C07227=1039.766,-84.411,-76.368,168.767,36.325,156.840
C07228=1039.759,-84.660,-76.358,168.765,36.326,156.840
C07229=1039.754,-84.910,-76.347,168.762,36.326,156.840
C07230=1039.747,-85.160,-76.336,168.760,36.326,156.840
C07231=1039.741,-85.409,-76.325,168.757,36.326,156.840
C07232=1039.734,-85.659,-76.314,168.755,36.326,156.840
C07233=1039.728,-85.909,-76.304,168.752,36.326,156.840
C07234=1039.722,-86.158,-76.293,168.750,36.327,156.840
C07235=1039.716,-86.408,-76.282,168.747,36.327,156.840
C07236=1039.709,-86.658,-76.271,168.745,36.327,156.840
C07237=1039.704,-86.908,-76.261,168.742,36.327,156.840
C07238=1039.698,-87.158,-76.250,168.740,36.327,156.840
C07239=1039.691,-87.407,-76.240,168.737,36.327,156.840
C07240=1039.685,-87.656,-76.229,168.735,36.327,156.840
C07241=1039.679,-87.907,-76.218,168.732,36.327,156.840
C07242=1039.673,-88.156,-76.207,168.730,36.327,156.840
C07243=1039.667,-88.405,-76.196,168.727,36.328,156.840
C07244=1039.660,-88.655,-76.186,168.725,36.328,156.840
C07245=1039.654,-88.905,-76.176,168.722,36.328,156.840
C07246=1039.649,-89.155,-76.165,168.720,36.328,156.840
C07247=1039.642,-89.405,-76.154,168.717,36.328,156.840
C07248=1039.636,-89.654,-76.143,168.715,36.328,156.840
C07249=1039.630,-89.904,-76.132,168.712,36.328,156.840
C07250=1039.624,-90.153,-76.123,168.710,36.328,156.840
C07251=1039.618,-90.404,-76.111,168.707,36.328,156.840
C07252=1039.611,-90.653,-76.101,168.705,36.329,156.841
C07253=1039.605,-90.902,-76.090,168.702,36.329,156.841
C07254=1039.600,-91.152,-76.080,168.700,36.329,156.841
C07255=1039.593,-91.402,-76.069,168.697,36.329,156.841
C07256=1039.587,-91.652,-76.059,168.695,36.330,156.841
C07257=1039.581,-91.901,-76.048,168.692,36.330,156.841
C07258=1039.575,-92.151,-76.038,168.690,36.330,156.841
C07259=1039.569,-92.401,-76.027,168.687,36.330,156.841
C07260=1039.562,-92.650,-76.017,168.685,36.330,156.841
C07261=1039.557,-92.901,-76.006,168.682,36.330,156.841
C07262=1039.550,-93.150,-75.996,168.680,36.330,156.841
C07263=1039.545,-93.399,-75.985,168.678,36.331,156.841
C07264=1039.539,-93.650,-75.975,168.676,36.331,156.841
C07265=1039.532,-93.899,-75.965,168.673,36.331,156.841
C07266=1039.526,-94.149,-75.954,168.671,36.331,156.841
C07267=1039.520,-94.399,-75.944,168.668,36.331,156.841
C07268=1039.515,-94.648,-75.933,168.666,36.331,156.841
C07269=1039.508,-94.897,-75.923,168.663,36.331,156.841
C07270=1039.502,-95.148,-75.912,168.661,36.332,156.841
C07271=1039.496,-95.398,-75.901,168.658,36.332,156.841
C07272=1039.490,-95.647,-75.891,168.656,36.332,156.841
C07273=1039.484,-95.897,-75.881,168.653,36.333,156.841
C07274=1039.478,-96.146,-75.871,168.651,36.333,156.841
C07275=1039.472,-96.396,-75.861,168.648,36.333,156.841
C07276=1039.466,-96.645,-75.850,168.646,36.333,156.841
C07277=1039.460,-96.896,-75.840,168.643,36.333,156.841
C07278=1039.454,-97.146,-75.829,168.641,36.333,156.841
C07279=1039.448,-97.395,-75.819,168.638,36.333,156.841
C07280=1039.442,-97.645,-75.809,168.636,36.334,156.842
C07281=1039.436,-97.895,-75.799,168.633,36.334,156.842
C07282=1039.430,-98.144,-75.789,168.630,36.335,156.842
C07283=1039.423,-98.394,-75.779,168.628,36.335,156.842
C07284=1039.417,-98.644,-75.768,168.625,36.335,156.842
C07285=1039.411,-98.894,-75.758,168.623,36.335,156.842
C07286=1039.404,-99.143,-75.748,168.620,36.336,156.842
C07287=1039.399,-99.393,-75.738,168.618,36.336,156.842
C07288=1039.392,-99.680,-75.727,168.615,36.336,156.842
C07289=1039.384,-99.967,-75.715,168.612,36.337,156.842
C07290=1039.378,-100.255,-75.703,168.609,36.337,156.842
C07291=1039.371,-100.541,-75.692,168.606,36.338,156.842
C07292=1039.364,-100.791,-75.681,168.603,36.338,156.842
C07293=1039.358,-101.041,-75.671,168.601,36.338,156.842
C07294=1039.352,-101.291,-75.662,168.598,36.338,156.842
C07295=1039.346,-101.540,-75.651,168.596,36.339,156.842
C07296=1039.340,-101.790,-75.641,168.593,36.340,156.843
C07297=1039.334,-102.040,-75.632,168.591,36.340,156.843
C07298=1039.328,-102.289,-75.621,168.589,36.340,156.843
C07299=1039.322,-102.539,-75.611,168.586,36.340,156.843
C07300=1039.316,-102.789,-75.602,168.584,36.341,156.843
C07301=1039.310,-103.038,-75.591,168.581,36.341,156.843
C07302=1039.303,-103.288,-75.582,168.579,36.342,156.843
C07303=1039.298,-103.538,-75.572,168.576,36.341,156.843
C07304=1039.291,-103.787,-75.561,168.574,36.342,156.843
C07305=1039.285,-104.037,-75.552,168.571,36.343,156.843
C07306=1039.279,-104.287,-75.542,168.568,36.343,156.843
C07307=1039.274,-104.537,-75.532,168.566,36.343,156.843
C07308=1039.267,-104.786,-75.522,168.563,36.343,156.843
C07309=1039.261,-105.036,-75.512,168.561,36.344,156.843
C07310=1039.255,-105.286,-75.503,168.558,36.345,156.844
C07311=1039.249,-105.536,-75.492,168.556,36.345,156.844
C07312=1039.243,-105.786,-75.483,168.553,36.345,156.844
C07313=1039.237,-106.035,-75.472,168.550,36.345,156.844
C07314=1039.231,-106.285,-75.463,168.548,36.346,156.844
C07315=1039.224,-106.535,-75.453,168.545,36.347,156.844
C07316=1039.219,-106.785,-75.443,168.543,36.347,156.844
C07317=1039.213,-107.034,-75.434,168.540,36.347,156.844
C07318=1039.207,-107.284,-75.424,168.538,36.348,156.844
C07319=1039.200,-107.533,-75.414,168.535,36.348,156.844
C07320=1039.194,-107.783,-75.404,168.532,36.349,156.844
C07321=1039.188,-108.033,-75.395,168.530,36.349,156.844
C07322=1039.182,-108.283,-75.384,168.528,36.350,156.844
C07323=1039.176,-108.533,-75.375,168.526,36.350,156.844
C07324=1039.170,-108.783,-75.365,168.523,36.350,156.845
C07325=1039.164,-109.033,-75.356,168.520,36.351,156.845
C07326=1039.158,-109.282,-75.346,168.518,36.352,156.845
C07327=1039.152,-109.532,-75.337,168.515,36.352,156.845
C07328=1039.146,-109.781,-75.327,168.513,36.352,156.845
C07329=1039.140,-110.031,-75.318,168.510,36.353,156.845
C07330=1039.134,-110.281,-75.308,168.507,36.354,156.845
C07331=1039.127,-110.531,-75.299,168.505,36.354,156.845
C07332=1039.121,-110.780,-75.289,168.502,36.354,156.845
///RCONF 1,0,0,0,1,0,0,0,0,0,0,0,0,0,0,0,0,0,0,0,0,0,0,0
C07333=1039.115,-111.030,-75.280,168.499,36.355,156.845
C07334=1039.109,-111.280,-75.270,168.497,36.356,156.845
C07335=1039.103,-111.530,-75.260,168.494,36.356,156.846
C07336=1039.097,-111.780,-75.251,168.492,36.356,156.846
C07337=1039.090,-112.029,-75.241,168.489,36.357,156.846
C07338=1039.086,-112.279,-75.232,168.486,36.357,156.846
C07339=1039.079,-112.529,-75.222,168.484,36.358,156.846
C07340=1039.073,-112.778,-75.212,168.481,36.359,156.846
C07341=1039.067,-113.028,-75.203,168.479,36.359,156.846
C07342=1039.061,-113.278,-75.193,168.477,36.359,156.846
C07343=1039.055,-113.528,-75.184,168.474,36.360,156.846
C07344=1039.049,-113.778,-75.174,168.472,36.361,156.846
C07345=1039.043,-114.027,-75.165,168.469,36.361,156.847
C07346=1039.037,-114.276,-75.155,168.467,36.362,156.847
C07347=1039.031,-114.526,-75.146,168.464,36.362,156.847
C07348=1039.025,-114.777,-75.137,168.461,36.363,156.847
C07349=1039.019,-115.027,-75.127,168.459,36.363,156.847
C07350=1039.012,-115.276,-75.118,168.456,36.364,156.847
C07351=1039.007,-115.525,-75.109,168.453,36.365,156.847
C07352=1038.999,-115.812,-75.098,168.450,36.365,156.847
C07353=1038.993,-116.098,-75.087,168.447,36.366,156.847
C07354=1038.985,-116.385,-75.077,168.444,36.367,156.847
C07355=1038.979,-116.671,-75.066,168.441,36.367,156.848
C07356=1038.972,-116.921,-75.057,168.439,36.368,156.848
C07357=1038.967,-117.170,-75.048,168.436,36.368,156.848
C07358=1038.961,-117.420,-75.038,168.434,36.369,156.848
C07359=1038.954,-117.670,-75.028,168.432,36.370,156.848
C07360=1038.949,-117.920,-75.020,168.429,36.370,156.848
C07361=1038.942,-118.169,-75.011,168.427,36.371,156.848
C07362=1038.936,-118.419,-75.001,168.424,36.372,156.848
C07363=1038.930,-118.669,-74.993,168.421,36.372,156.848
C07364=1038.924,-118.919,-74.983,168.419,36.373,156.849
C07365=1038.918,-119.168,-74.974,168.416,36.374,156.849
C07366=1038.912,-119.418,-74.964,168.413,36.374,156.849
C07367=1038.906,-119.668,-74.955,168.411,36.375,156.849
C07368=1038.900,-119.918,-74.946,168.408,36.376,156.849
C07369=1038.894,-120.167,-74.937,168.405,36.376,156.849
C07370=1038.888,-120.417,-74.928,168.403,36.377,156.849
C07371=1038.882,-120.667,-74.919,168.400,36.378,156.849
C07372=1038.876,-120.917,-74.909,168.398,36.378,156.849
C07373=1038.870,-121.167,-74.901,168.395,36.379,156.850
C07374=1038.864,-121.416,-74.892,168.393,36.379,156.850
C07375=1038.858,-121.666,-74.883,168.391,36.380,156.850
C07376=1038.852,-121.916,-74.874,168.388,36.381,156.850
C07377=1038.846,-122.165,-74.864,168.385,36.381,156.850
C07378=1038.840,-122.416,-74.855,168.383,36.382,156.850
C07379=1038.834,-122.665,-74.847,168.380,36.383,156.850
C07380=1038.828,-122.915,-74.838,168.377,36.384,156.851
C07381=1038.822,-123.165,-74.828,168.375,36.385,156.851
C07382=1038.816,-123.414,-74.819,168.372,36.385,156.851
C07383=1038.810,-123.664,-74.811,168.369,36.386,156.851
C07384=1038.803,-123.914,-74.801,168.367,36.387,156.851
C07385=1038.798,-124.163,-74.793,168.364,36.387,156.851
C07386=1038.792,-124.413,-74.783,168.361,36.388,156.851
C07387=1038.785,-124.663,-74.775,168.359,36.389,156.851
C07388=1038.780,-124.912,-74.766,168.357,36.389,156.851
C07389=1038.774,-125.163,-74.757,168.354,36.391,156.852
C07390=1038.767,-125.412,-74.748,168.352,36.391,156.852
C07391=1038.762,-125.662,-74.739,168.349,36.392,156.852
C07392=1038.756,-125.912,-74.730,168.346,36.392,156.852
C07393=1038.750,-126.161,-74.722,168.344,36.393,156.852
C07394=1038.744,-126.412,-74.713,168.341,36.394,156.852
C07395=1038.738,-126.661,-74.704,168.338,36.395,156.852
C07396=1038.732,-126.911,-74.696,168.336,36.396,156.853
C07397=1038.725,-127.161,-74.686,168.333,36.396,156.853
C07398=1038.720,-127.410,-74.678,168.330,36.397,156.853
C07399=1038.714,-127.661,-74.669,168.328,36.398,156.853
C07400=1038.708,-127.910,-74.660,168.326,36.399,156.853
C07401=1038.703,-128.160,-74.650,168.324,36.399,156.853
C07402=1038.698,-128.409,-74.640,168.321,36.399,156.853
C07403=1038.695,-128.658,-74.630,168.318,36.398,156.853
C07404=1038.692,-128.909,-74.618,168.316,36.397,156.853
C07405=1038.690,-129.158,-74.607,168.314,36.396,156.853
C07406=1038.689,-129.409,-74.594,168.312,36.394,156.852
C07407=1038.689,-129.658,-74.581,168.311,36.391,156.852
C07408=1038.690,-129.909,-74.567,168.308,36.388,156.851
C07409=1038.690,-130.159,-74.553,168.307,36.384,156.851
C07410=1038.692,-130.409,-74.538,168.306,36.381,156.850
C07411=1038.695,-130.659,-74.523,168.304,36.377,156.849
C07412=1038.698,-130.909,-74.507,168.303,36.372,156.849
C07413=1038.703,-131.160,-74.490,168.301,36.367,156.848
C07414=1038.707,-131.409,-74.473,168.301,36.361,156.847
C07415=1038.713,-131.660,-74.455,168.300,36.355,156.846
C07416=1038.372,-131.683,-74.721,168.252,36.557,156.880
C07417=1038.366,-131.435,-74.739,168.253,36.564,156.881
C07418=1038.360,-131.184,-74.756,168.254,36.569,156.882
C07419=1038.356,-130.934,-74.773,168.255,36.574,156.883
C07420=1038.353,-130.683,-74.788,168.256,36.579,156.883
C07421=1038.350,-130.434,-74.805,168.258,36.584,156.884
C07422=1038.348,-130.184,-74.819,168.259,36.587,156.885
C07423=1038.347,-129.933,-74.834,168.261,36.591,156.885
C07424=1038.346,-129.683,-74.847,168.263,36.593,156.886
C07425=1038.347,-129.433,-74.860,168.264,36.596,156.886
C07426=1038.349,-129.184,-74.873,168.266,36.598,156.887
C07427=1038.350,-128.934,-74.885,168.269,36.600,156.887
C07428=1038.352,-128.683,-74.896,168.271,36.601,156.887
C07429=1038.357,-128.434,-74.907,168.273,36.601,156.887
C07430=1038.361,-128.184,-74.917,168.276,36.602,156.887
C07431=1038.365,-127.934,-74.926,168.278,36.601,156.887
C07432=1038.371,-127.685,-74.935,168.281,36.601,156.887
C07433=1038.377,-127.435,-74.944,168.283,36.600,156.887
C07434=1038.383,-127.185,-74.953,168.286,36.599,156.887
C07435=1038.389,-126.935,-74.962,168.288,36.598,156.887
C07436=1038.395,-126.686,-74.970,168.291,36.597,156.887
C07437=1038.401,-126.436,-74.979,168.293,36.597,156.886
C07438=1038.407,-126.185,-74.988,168.296,36.596,156.886
C07439=1038.413,-125.937,-74.997,168.299,36.595,156.886
C07440=1038.419,-125.686,-75.005,168.301,36.594,156.886
C07441=1038.425,-125.437,-75.015,168.304,36.593,156.886
C07442=1038.431,-125.187,-75.023,168.307,36.593,156.886
C07443=1038.437,-124.937,-75.032,168.309,36.592,156.886
C07444=1038.443,-124.688,-75.041,168.312,36.591,156.885
C07445=1038.450,-124.438,-75.050,168.315,36.590,156.885
C07446=1038.455,-124.188,-75.059,168.317,36.589,156.885
C07447=1038.461,-123.939,-75.068,168.320,36.589,156.885
C07448=1038.467,-123.688,-75.077,168.322,36.588,156.885
C07449=1038.474,-123.439,-75.086,168.324,36.587,156.885
C07450=1038.479,-123.189,-75.094,168.327,36.587,156.885
C07451=1038.485,-122.939,-75.104,168.330,36.585,156.885
C07452=1038.491,-122.689,-75.113,168.332,36.585,156.884
C07453=1038.497,-122.440,-75.122,168.335,36.584,156.884
C07454=1038.504,-122.190,-75.131,168.338,36.583,156.884
C07455=1038.509,-121.940,-75.140,168.340,36.583,156.884
C07456=1038.515,-121.691,-75.149,168.343,36.582,156.884
C07457=1038.521,-121.440,-75.158,168.346,36.581,156.884
C07458=1038.527,-121.190,-75.167,168.348,36.581,156.884
C07459=1038.533,-120.942,-75.176,168.351,36.580,156.884
C07460=1038.539,-120.691,-75.185,168.354,36.579,156.884
C07461=1038.545,-120.441,-75.194,168.355,36.578,156.883
C07462=1038.551,-120.192,-75.204,168.358,36.577,156.883
C07463=1038.557,-119.942,-75.212,168.361,36.577,156.883
C07464=1038.563,-119.692,-75.222,168.363,36.576,156.883
C07465=1038.570,-119.443,-75.231,168.366,36.575,156.883
C07466=1038.575,-119.193,-75.239,168.369,36.575,156.883
C07467=1038.581,-118.943,-75.249,168.371,36.574,156.883
C07468=1038.587,-118.693,-75.259,168.374,36.573,156.883
C07469=1038.593,-118.443,-75.267,168.377,36.573,156.882
C07470=1038.599,-118.194,-75.277,168.379,36.572,156.882
C07471=1038.605,-117.944,-75.286,168.382,36.571,156.882
C07472=1038.612,-117.694,-75.295,168.385,36.571,156.882
C07473=1038.618,-117.444,-75.304,168.387,36.570,156.882
C07474=1038.623,-117.195,-75.313,168.390,36.569,156.882
C07475=1038.630,-116.945,-75.323,168.392,36.569,156.882
C07476=1038.636,-116.695,-75.332,168.394,36.568,156.882
C07477=1038.642,-116.409,-75.343,168.397,36.567,156.882
C07478=1038.650,-116.122,-75.354,168.400,36.567,156.881
C07479=1038.657,-115.836,-75.364,168.403,36.566,156.881
C07480=1038.663,-115.550,-75.375,168.406,36.565,156.881
C07481=1038.670,-115.300,-75.384,168.409,36.565,156.881
C07482=1038.676,-115.051,-75.393,168.412,36.564,156.881
C07483=1038.682,-114.801,-75.403,168.414,36.563,156.881
C07484=1038.688,-114.550,-75.412,168.417,36.563,156.881
C07485=1038.694,-114.301,-75.421,168.420,36.562,156.881
C07486=1038.700,-114.052,-75.431,168.422,36.562,156.881
C07487=1038.706,-113.802,-75.440,168.425,36.561,156.880
C07488=1038.712,-113.552,-75.450,168.427,36.560,156.880
C07489=1038.718,-113.302,-75.459,168.430,36.560,156.880
C07490=1038.724,-113.052,-75.469,168.433,36.560,156.880
C07491=1038.730,-112.803,-75.478,168.434,36.559,156.880
C07492=1038.736,-112.553,-75.488,168.437,36.558,156.880
C07493=1038.742,-112.304,-75.497,168.440,36.558,156.880
C07494=1038.748,-112.054,-75.507,168.442,36.557,156.880
C07495=1038.753,-111.803,-75.516,168.445,36.556,156.880
C07496=1038.760,-111.553,-75.526,168.447,36.556,156.880
C07497=1038.766,-111.304,-75.535,168.450,36.556,156.880
C07498=1038.772,-111.054,-75.545,168.453,36.555,156.880
C07499=1038.778,-110.804,-75.554,168.455,36.554,156.879
C07500=1038.784,-110.555,-75.564,168.458,36.554,156.879
C07501=1038.790,-110.305,-75.573,168.461,36.553,156.879
C07502=1038.796,-110.055,-75.583,168.463,36.553,156.879
C07503=1038.802,-109.805,-75.592,168.466,36.552,156.879
C07504=1038.809,-109.556,-75.603,168.468,36.552,156.879
C07505=1038.815,-109.306,-75.612,168.471,36.551,156.879
C07506=1038.821,-109.057,-75.622,168.474,36.550,156.879
///RCONF 1,0,0,0,0,0,0,0,0,0,0,0,0,0,0,0,0,0,0,0,0,0,0,0
C07507=1038.827,-108.807,-75.631,168.476,36.550,156.879
C07508=1038.833,-108.557,-75.641,168.479,36.550,156.879
C07509=1038.840,-108.307,-75.651,168.481,36.549,156.879
C07510=1038.845,-108.057,-75.661,168.483,36.548,156.878
C07511=1038.851,-107.807,-75.670,168.486,36.548,156.878
C07512=1038.857,-107.558,-75.680,168.488,36.548,156.878
C07513=1038.864,-107.308,-75.689,168.491,36.547,156.878
C07514=1038.870,-107.058,-75.699,168.494,36.546,156.878
C07515=1038.876,-106.810,-75.709,168.496,36.546,156.878
C07516=1038.882,-106.560,-75.718,168.499,36.546,156.878
C07517=1038.887,-106.310,-75.729,168.501,36.545,156.878
C07518=1038.893,-106.060,-75.738,168.504,36.544,156.878
C07519=1038.900,-105.810,-75.748,168.507,36.544,156.878
C07520=1038.906,-105.560,-75.757,168.509,36.544,156.878
C07521=1038.911,-105.311,-75.768,168.512,36.543,156.878
C07522=1038.918,-105.061,-75.778,168.514,36.543,156.878
C07523=1038.924,-104.811,-75.787,168.517,36.542,156.877
C07524=1038.930,-104.561,-75.797,168.520,36.542,156.877
C07525=1038.936,-104.312,-75.808,168.522,36.542,156.877
C07526=1038.942,-104.062,-75.817,168.525,36.541,156.877
C07527=1038.948,-103.812,-75.827,168.527,36.541,156.877
C07528=1038.954,-103.562,-75.836,168.530,36.540,156.877
C07529=1038.960,-103.313,-75.847,168.532,36.540,156.877
C07530=1038.966,-103.063,-75.857,168.535,36.540,156.877
C07531=1038.972,-102.813,-75.866,168.537,36.539,156.877
C07532=1038.979,-102.564,-75.877,168.539,36.539,156.877
C07533=1038.985,-102.313,-75.887,168.542,36.538,156.877
C07534=1038.991,-102.064,-75.897,168.544,36.538,156.877
C07535=1038.997,-101.814,-75.906,168.547,36.538,156.877
C07536=1039.003,-101.564,-75.917,168.550,36.537,156.877
C07537=1039.009,-101.314,-75.927,168.552,36.537,156.877
C07538=1039.016,-101.065,-75.937,168.555,36.536,156.876
C07539=1039.022,-100.816,-75.947,168.557,36.536,156.876
C07540=1039.027,-100.565,-75.957,168.560,36.536,156.876
C07541=1039.035,-100.279,-75.969,168.563,36.535,156.876
C07542=1039.042,-99.991,-75.980,168.566,36.534,156.876
C07543=1039.049,-99.704,-75.992,168.569,36.534,156.876
C07544=1039.055,-99.417,-76.003,168.572,36.534,156.876
C07545=1039.062,-99.167,-76.013,168.574,36.534,156.876
C07546=1039.068,-98.917,-76.024,168.577,36.533,156.876
C07547=1039.074,-98.668,-76.034,168.579,36.532,156.876
C07548=1039.081,-98.418,-76.043,168.582,36.532,156.876
C07549=1039.086,-98.168,-76.054,168.585,36.532,156.876
C07550=1039.092,-97.919,-76.064,168.587,36.532,156.876
C07551=1039.099,-97.669,-76.073,168.590,36.531,156.875
C07552=1039.105,-97.419,-76.085,168.592,36.531,156.875
C07553=1039.111,-97.169,-76.094,168.595,36.531,156.875
C07554=1039.117,-96.920,-76.105,168.597,36.531,156.875
C07555=1039.123,-96.670,-76.115,168.600,36.531,156.875
C07556=1039.129,-96.420,-76.126,168.602,36.530,156.875
C07557=1039.135,-96.171,-76.136,168.605,36.530,156.875
C07558=1039.141,-95.921,-76.146,168.607,36.530,156.875
C07559=1039.146,-95.672,-76.157,168.609,36.529,156.875
C07560=1039.153,-95.421,-76.167,168.611,36.529,156.875
C07561=1039.159,-95.172,-76.178,168.614,36.529,156.875
C07562=1039.165,-94.922,-76.188,168.617,36.529,156.875
C07563=1039.171,-94.672,-76.198,168.619,36.529,156.875
C07564=1039.177,-94.423,-76.209,168.622,36.529,156.875
C07565=1039.183,-94.174,-76.219,168.624,36.528,156.875
C07566=1039.189,-93.923,-76.230,168.627,36.528,156.875
C07567=1039.196,-93.674,-76.240,168.629,36.528,156.875
C07568=1039.201,-93.423,-76.250,168.632,36.527,156.875
C07569=1039.207,-93.174,-76.261,168.634,36.527,156.875
C07570=1039.213,-92.925,-76.271,168.637,36.527,156.875
C07571=1039.219,-92.675,-76.282,168.639,36.527,156.875
C07572=1039.226,-92.425,-76.292,168.642,36.527,156.875
C07573=1039.231,-92.175,-76.303,168.644,36.527,156.875
C07574=1039.238,-91.926,-76.313,168.647,36.526,156.875
C07575=1039.243,-91.676,-76.324,168.649,36.526,156.875
C07576=1039.250,-91.426,-76.335,168.652,36.526,156.875
C07577=1039.256,-91.177,-76.345,168.654,36.525,156.874
C07578=1039.262,-90.927,-76.356,168.657,36.525,156.874
C07579=1039.268,-90.677,-76.366,168.659,36.525,156.874
C07580=1039.274,-90.427,-76.377,168.662,36.525,156.874
C07581=1039.280,-90.178,-76.388,168.664,36.525,156.874
C07582=1039.287,-89.929,-76.398,168.667,36.525,156.874
C07583=1039.292,-89.678,-76.408,168.669,36.525,156.874
C07584=1039.299,-89.429,-76.419,168.672,36.524,156.874
C07585=1039.305,-89.179,-76.430,168.674,36.524,156.874
C07586=1039.311,-88.930,-76.440,168.677,36.524,156.874
C07587=1039.318,-88.680,-76.451,168.680,36.523,156.874
C07588=1039.323,-88.430,-76.461,168.682,36.523,156.874
C07589=1039.329,-88.180,-76.472,168.685,36.523,156.874
C07590=1039.335,-87.931,-76.482,168.687,36.523,156.874
C07591=1039.342,-87.681,-76.494,168.690,36.523,156.874
C07592=1039.348,-87.432,-76.504,168.692,36.523,156.874
C07593=1039.354,-87.182,-76.515,168.695,36.523,156.874
C07594=1039.360,-86.932,-76.526,168.697,36.523,156.874
C07595=1039.366,-86.682,-76.536,168.700,36.522,156.874
C07596=1039.372,-86.433,-76.547,168.702,36.522,156.874
C07597=1039.379,-86.182,-76.558,168.705,36.522,156.874
C07598=1039.385,-85.933,-76.568,168.707,36.522,156.874
C07599=1039.391,-85.683,-76.579,168.710,36.521,156.874
C07600=1039.397,-85.434,-76.590,168.712,36.521,156.874
C07601=1039.404,-85.184,-76.600,168.715,36.521,156.874
C07602=1039.410,-84.934,-76.612,168.717,36.521,156.874
C07603=1039.416,-84.685,-76.623,168.720,36.521,156.874
C07604=1039.422,-84.436,-76.633,168.722,36.521,156.874
C07605=1039.429,-84.150,-76.645,168.725,36.521,156.874
C07606=1039.437,-83.865,-76.657,168.728,36.521,156.874
C07607=1039.444,-83.580,-76.669,168.731,36.520,156.874
C07608=1039.450,-83.295,-76.683,168.733,36.520,156.874
C07609=1039.457,-83.046,-76.693,168.736,36.520,156.874
C07610=1039.463,-82.796,-76.705,168.738,36.520,156.874
C07611=1039.469,-82.546,-76.715,168.741,36.520,156.874
C07612=1039.476,-82.296,-76.726,168.742,36.519,156.873
C07613=1039.482,-82.047,-76.737,168.745,36.519,156.873
C07614=1039.488,-81.797,-76.748,168.747,36.519,156.873
C07615=1039.495,-81.548,-76.758,168.750,36.519,156.873
C07616=1039.501,-81.297,-76.770,168.752,36.519,156.873
C07617=1039.507,-81.048,-76.781,168.755,36.519,156.873
C07618=1039.513,-80.799,-76.791,168.757,36.519,156.873
C07619=1039.519,-80.548,-76.802,168.760,36.519,156.873
C07620=1039.525,-80.299,-76.813,168.762,36.519,156.873
C07621=1039.532,-80.049,-76.824,168.765,36.519,156.873
C07622=1039.538,-79.800,-76.835,168.767,36.518,156.873
C07623=1039.545,-79.550,-76.847,168.770,36.518,156.873
C07624=1039.550,-79.301,-76.857,168.772,36.518,156.873
C07625=1039.557,-79.050,-76.869,168.775,36.518,156.873
C07626=1039.563,-78.801,-76.880,168.777,36.518,156.873
C07627=1039.569,-78.551,-76.891,168.780,36.518,156.873
C07628=1039.575,-78.302,-76.902,168.782,36.518,156.873
C07629=1039.581,-78.052,-76.914,168.784,36.518,156.873
C07630=1039.587,-77.802,-76.924,168.787,36.518,156.873
C07631=1039.593,-77.552,-76.936,168.789,36.518,156.873
C07632=1039.600,-77.303,-76.947,168.792,36.518,156.873
C07633=1039.606,-77.053,-76.958,168.794,36.518,156.873
C07634=1039.612,-76.804,-76.969,168.797,36.518,156.873
C07635=1039.619,-76.553,-76.980,168.799,36.518,156.873
C07636=1039.625,-76.305,-76.992,168.802,36.518,156.873
C07637=1039.631,-76.054,-77.003,168.804,36.518,156.873
C07638=1039.637,-75.805,-77.014,168.806,36.518,156.873
C07639=1039.643,-75.555,-77.026,168.809,36.518,156.873
C07640=1039.649,-75.306,-77.037,168.811,36.518,156.873
C07641=1039.655,-75.056,-77.048,168.814,36.519,156.873
C07642=1039.662,-74.806,-77.060,168.816,36.519,156.873
C07643=1039.668,-74.557,-77.071,168.819,36.519,156.873
C07644=1039.674,-74.306,-77.082,168.821,36.519,156.873
C07645=1039.680,-74.058,-77.094,168.823,36.519,156.873
C07646=1039.686,-73.807,-77.105,168.826,36.519,156.873
C07647=1039.692,-73.558,-77.116,168.828,36.519,156.873
C07648=1039.699,-73.308,-77.128,168.831,36.519,156.873
C07649=1039.704,-73.058,-77.139,168.833,36.519,156.873
C07650=1039.711,-72.809,-77.151,168.835,36.519,156.873
C07651=1039.717,-72.559,-77.162,168.838,36.519,156.873
C07652=1039.723,-72.310,-77.174,168.840,36.519,156.873
C07653=1039.729,-72.059,-77.186,168.843,36.519,156.873
C07654=1039.735,-71.811,-77.197,168.846,36.520,156.874
C07655=1039.741,-71.560,-77.209,168.848,36.520,156.874
C07656=1039.747,-71.311,-77.220,168.851,36.520,156.874
C07657=1039.753,-71.061,-77.231,168.853,36.520,156.874
C07658=1039.759,-70.811,-77.244,168.856,36.520,156.874
C07659=1039.765,-70.562,-77.255,168.858,36.521,156.874
C07660=1039.772,-70.312,-77.267,168.860,36.521,156.874
C07661=1039.777,-70.063,-77.278,168.863,36.521,156.874
C07662=1039.783,-69.813,-77.290,168.865,36.521,156.874
C07663=1039.790,-69.563,-77.301,168.867,36.521,156.874
C07664=1039.796,-69.314,-77.313,168.870,36.521,156.874
C07665=1039.802,-69.064,-77.324,168.872,36.521,156.874
C07666=1039.807,-68.814,-77.336,168.875,36.521,156.874
C07667=1039.814,-68.565,-77.348,168.877,36.522,156.874
C07668=1039.820,-68.315,-77.360,168.879,36.522,156.874
C07669=1039.827,-68.032,-77.373,168.882,36.522,156.874
C07670=1039.834,-67.750,-77.386,168.885,36.523,156.874
C07671=1039.841,-67.467,-77.400,168.887,36.523,156.874
C07672=1039.848,-67.184,-77.413,168.890,36.523,156.874
C07673=1039.855,-66.934,-77.425,168.892,36.523,156.874
C07674=1039.860,-66.685,-77.436,168.895,36.523,156.874
C07675=1039.866,-66.435,-77.448,168.897,36.523,156.874
C07676=1039.873,-66.185,-77.460,168.900,36.523,156.874
C07677=1039.878,-65.936,-77.472,168.902,36.523,156.874
C07678=1039.885,-65.686,-77.484,168.904,36.524,156.874
C07679=1039.891,-65.436,-77.495,168.907,36.524,156.874
C07680=1039.897,-65.187,-77.506,168.909,36.524,156.874
C07681=1039.903,-64.937,-77.519,168.911,36.524,156.874
C07682=1039.910,-64.688,-77.531,168.914,36.524,156.874
C07683=1039.916,-64.437,-77.542,168.916,36.524,156.874
C07684=1039.921,-64.188,-77.554,168.918,36.524,156.874
C07685=1039.928,-63.939,-77.566,168.921,36.525,156.875
C07686=1039.935,-63.689,-77.578,168.923,36.525,156.875
C07687=1039.941,-63.439,-77.589,168.925,36.525,156.875
C07688=1039.946,-63.190,-77.602,168.928,36.526,156.875
C07689=1039.953,-62.940,-77.614,168.930,36.526,156.875
C07690=1039.960,-62.691,-77.626,168.933,36.526,156.875
C07691=1039.965,-62.441,-77.638,168.935,36.526,156.875
C07692=1039.971,-62.191,-77.649,168.937,36.526,156.875
C07693=1039.978,-61.942,-77.661,168.940,36.526,156.875
C07694=1039.984,-61.692,-77.673,168.942,36.526,156.875
C07695=1039.990,-61.442,-77.685,168.944,36.527,156.875
C07696=1039.997,-61.193,-77.697,168.947,36.527,156.875
C07697=1040.003,-60.944,-77.709,168.949,36.527,156.875
C07698=1040.009,-60.693,-77.721,168.951,36.528,156.875
C07699=1040.015,-60.444,-77.733,168.954,36.528,156.875
C07700=1040.022,-60.194,-77.745,168.956,36.528,156.875
C07701=1040.028,-59.944,-77.757,168.958,36.528,156.875
C07702=1040.035,-59.695,-77.769,168.961,36.528,156.875
C07703=1040.041,-59.446,-77.781,168.963,36.528,156.875
C07704=1040.046,-59.196,-77.793,168.966,36.529,156.875
C07705=1040.053,-58.946,-77.805,168.969,36.529,156.875
C07706=1040.059,-58.696,-77.817,168.971,36.529,156.875
C07707=1040.065,-58.446,-77.829,168.973,36.530,156.875
C07708=1040.072,-58.197,-77.841,168.976,36.530,156.875
C07709=1040.079,-57.947,-77.853,168.978,36.530,156.875
C07710=1040.084,-57.698,-77.865,168.980,36.530,156.875
C07711=1040.091,-57.448,-77.877,168.983,36.530,156.875
C07712=1040.097,-57.199,-77.889,168.985,36.530,156.875
C07713=1040.103,-56.949,-77.902,168.987,36.531,156.876
C07714=1040.110,-56.699,-77.914,168.990,36.531,156.876
C07715=1040.116,-56.450,-77.926,168.992,36.531,156.876
C07716=1040.122,-56.200,-77.938,168.994,36.532,156.876
C07717=1040.129,-55.935,-77.951,168.997,36.532,156.876
C07718=1040.136,-55.671,-77.963,168.999,36.532,156.876
C07719=1040.143,-55.405,-77.977,169.002,36.532,156.876
C07720=1040.150,-55.141,-77.990,169.004,36.532,156.876
C07721=1040.156,-54.891,-78.002,169.007,36.533,156.876
C07722=1040.162,-54.641,-78.015,169.009,36.533,156.876
C07723=1040.169,-54.392,-78.027,169.011,36.533,156.876
C07724=1040.175,-54.142,-78.039,169.014,36.533,156.876
C07725=1040.181,-53.892,-78.051,169.016,36.533,156.876
C07726=1040.188,-53.643,-78.063,169.018,36.533,156.876
C07727=1040.194,-53.393,-78.076,169.021,36.534,156.876
C07728=1040.201,-53.143,-78.088,169.023,36.534,156.876
C07729=1040.207,-52.894,-78.099,169.025,36.535,156.876
C07730=1040.213,-52.644,-78.112,169.028,36.535,156.876
C07731=1040.220,-52.394,-78.124,169.030,36.535,156.876
C07732=1040.226,-52.145,-78.137,169.032,36.535,156.876
C07733=1040.233,-51.879,-78.149,169.035,36.535,156.876
C07734=1040.239,-51.613,-78.162,169.037,36.536,156.876
C07735=1040.247,-51.346,-78.176,169.040,36.536,156.876
C07736=1040.253,-51.080,-78.189,169.042,36.536,156.876
C07737=1040.260,-50.831,-78.201,169.044,36.537,156.877
C07738=1040.266,-50.581,-78.214,169.047,36.537,156.877
C07739=1040.272,-50.332,-78.226,169.049,36.537,156.877
C07740=1040.278,-50.082,-78.239,169.051,36.537,156.877
C07741=1040.284,-49.832,-78.251,169.053,36.538,156.877
C07742=1040.291,-49.583,-78.264,169.057,36.539,156.877
C07743=1040.297,-49.333,-78.276,169.059,36.539,156.877
C07744=1040.303,-49.083,-78.289,169.061,36.539,156.877
C07745=1040.309,-48.834,-78.302,169.063,36.539,156.877
C07746=1040.316,-48.584,-78.314,169.066,36.540,156.877
C07747=1040.322,-48.335,-78.327,169.068,36.541,156.877
C07748=1040.328,-48.085,-78.340,169.070,36.541,156.877
C07749=1040.334,-47.835,-78.353,169.072,36.541,156.877
C07750=1040.341,-47.586,-78.364,169.075,36.542,156.878
C07751=1040.347,-47.337,-78.378,169.077,36.542,156.878
C07752=1040.353,-47.087,-78.390,169.079,36.542,156.878
C07753=1040.359,-46.837,-78.403,169.081,36.542,156.878
C07754=1040.366,-46.588,-78.416,169.084,36.543,156.878
C07755=1040.372,-46.337,-78.428,169.086,36.544,156.878
C07756=1040.378,-46.087,-78.441,169.088,36.544,156.878
C07757=1040.384,-45.838,-78.454,169.090,36.544,156.878
C07758=1040.391,-45.589,-78.466,169.093,36.545,156.878
C07759=1040.397,-45.339,-78.480,169.095,36.545,156.878
C07760=1040.403,-45.089,-78.492,169.097,36.546,156.878
C07761=1040.409,-44.840,-78.505,169.099,36.546,156.878
C07762=1040.416,-44.591,-78.517,169.102,36.546,156.878
C07763=1040.422,-44.341,-78.530,169.104,36.547,156.878
C07764=1040.428,-44.091,-78.543,169.106,36.547,156.878
C07765=1040.434,-43.842,-78.556,169.109,36.548,156.879
C07766=1040.441,-43.593,-78.568,169.112,36.548,156.879
C07767=1040.447,-43.342,-78.581,169.114,36.548,156.879
C07768=1040.454,-43.093,-78.595,169.116,36.549,156.879
C07769=1040.459,-42.843,-78.607,169.118,36.550,156.879
C07770=1040.466,-42.594,-78.620,169.120,36.550,156.879
C07771=1040.472,-42.344,-78.632,169.123,36.550,156.879
C07772=1040.479,-42.095,-78.646,169.125,36.551,156.879
C07773=1040.484,-41.845,-78.658,169.127,36.551,156.879
C07774=1040.491,-41.596,-78.671,169.129,36.551,156.879
C07775=1040.497,-41.346,-78.685,169.132,36.552,156.879
C07776=1040.504,-41.096,-78.697,169.134,36.552,156.879
C07777=1040.510,-40.847,-78.710,169.136,36.553,156.879
C07778=1040.516,-40.597,-78.723,169.138,36.553,156.880
C07779=1040.522,-40.348,-78.736,169.140,36.553,156.880
C07780=1040.529,-40.097,-78.749,169.143,36.554,156.880
C07781=1040.536,-39.848,-78.762,169.145,36.555,156.880
C07782=1040.542,-39.599,-78.775,169.147,36.555,156.880
C07783=1040.548,-39.349,-78.788,169.149,36.555,156.880
C07784=1040.554,-39.100,-78.801,169.152,36.556,156.880
C07785=1040.561,-38.850,-78.814,169.154,36.556,156.880
C07786=1040.567,-38.600,-78.827,169.157,36.557,156.880
C07787=1040.573,-38.351,-78.840,169.159,36.557,156.880
C07788=1040.579,-38.101,-78.854,169.161,36.558,156.880
C07789=1040.585,-37.851,-78.866,169.163,36.558,156.881
C07790=1040.592,-37.602,-78.879,169.166,36.558,156.881
C07791=1040.598,-37.352,-78.893,169.168,36.559,156.881
C07792=1040.604,-37.102,-78.906,169.170,36.560,156.881
C07793=1040.610,-36.853,-78.919,169.172,36.560,156.881
C07794=1040.617,-36.604,-78.932,169.174,36.561,156.881
C07795=1040.623,-36.355,-78.945,169.177,36.562,156.881
C07796=1040.629,-36.104,-78.958,169.179,36.562,156.881
C07797=1040.636,-35.824,-78.973,169.181,36.562,156.881
C07798=1040.643,-35.542,-78.988,169.184,36.563,156.881
C07799=1040.651,-35.261,-79.003,169.186,36.564,156.881
C07800=1040.657,-34.980,-79.018,169.188,36.564,156.882
C07801=1040.664,-34.730,-79.032,169.191,36.565,156.882
C07802=1040.670,-34.481,-79.045,169.193,36.566,156.882
C07803=1040.676,-34.232,-79.058,169.196,36.566,156.882
C07804=1040.683,-33.982,-79.072,169.198,36.567,156.882
C07805=1040.689,-33.732,-79.084,169.200,36.567,156.882
C07806=1040.695,-33.483,-79.098,169.202,36.567,156.882
C07807=1040.701,-33.233,-79.111,169.205,36.568,156.882
C07808=1040.708,-32.983,-79.124,169.207,36.569,156.882
C07809=1040.714,-32.734,-79.138,169.209,36.569,156.883
C07810=1040.720,-32.485,-79.151,169.211,36.570,156.883
C07811=1040.727,-32.235,-79.165,169.213,36.571,156.883
C07812=1040.733,-31.986,-79.178,169.215,36.571,156.883
C07813=1040.740,-31.736,-79.191,169.218,36.571,156.883
C07814=1040.745,-31.486,-79.204,169.220,36.572,156.883
C07815=1040.752,-31.236,-79.218,169.222,36.573,156.883
C07816=1040.758,-30.987,-79.231,169.224,36.573,156.883
C07817=1040.764,-30.738,-79.244,169.226,36.574,156.883
C07818=1040.771,-30.488,-79.258,169.228,36.574,156.883
C07819=1040.777,-30.239,-79.271,169.230,36.574,156.883
C07820=1040.783,-29.989,-79.285,169.234,36.575,156.884
C07821=1040.790,-29.739,-79.298,169.236,36.576,156.884
C07822=1040.796,-29.490,-79.312,169.238,36.576,156.884
C07823=1040.803,-29.240,-79.325,169.240,36.577,156.884
C07824=1040.809,-28.991,-79.338,169.242,36.578,156.884
C07825=1040.815,-28.741,-79.352,169.244,36.578,156.884
C07826=1040.822,-28.491,-79.366,169.246,36.578,156.884
C07827=1040.828,-28.242,-79.379,169.249,36.579,156.884
C07828=1040.834,-27.993,-79.392,169.251,36.580,156.884
C07829=1040.841,-27.743,-79.406,169.253,36.580,156.884
C07830=1040.847,-27.494,-79.419,169.255,36.581,156.885
C07831=1040.854,-27.244,-79.433,169.257,36.581,156.885
C07832=1040.860,-26.994,-79.446,169.259,36.582,156.885
C07833=1040.866,-26.745,-79.460,169.261,36.583,156.885
C07834=1040.873,-26.495,-79.474,169.263,36.583,156.885
C07835=1040.879,-26.246,-79.488,169.267,36.584,156.885
C07836=1040.884,-25.997,-79.502,169.269,36.585,156.885
C07837=1040.891,-25.747,-79.515,169.271,36.585,156.885
C07838=1040.897,-25.497,-79.529,169.273,36.586,156.886
C07839=1040.904,-25.247,-79.543,169.275,36.587,156.886
C07840=1040.910,-24.998,-79.556,169.277,36.587,156.886
C07841=1040.916,-24.749,-79.571,169.279,36.588,156.886
C07842=1040.922,-24.499,-79.584,169.281,36.589,156.886
C07843=1040.929,-24.250,-79.598,169.283,36.589,156.886
C07844=1040.935,-23.999,-79.612,169.285,36.590,156.886
C07845=1040.941,-23.750,-79.625,169.288,36.590,156.886
C07846=1040.947,-23.501,-79.639,169.290,36.591,156.886
C07847=1040.953,-23.251,-79.653,169.292,36.592,156.887
C07848=1040.960,-23.002,-79.667,169.294,36.592,156.887
C07849=1040.966,-22.752,-79.680,169.297,36.593,156.887
C07850=1040.972,-22.503,-79.695,169.299,36.594,156.887
C07851=1040.979,-22.253,-79.708,169.301,36.594,156.887
C07852=1040.985,-22.003,-79.722,169.303,36.595,156.887
C07853=1040.991,-21.753,-79.736,169.305,36.596,156.887
C07854=1040.998,-21.505,-79.750,169.307,36.596,156.887
C07855=1041.004,-21.255,-79.764,169.309,36.597,156.888
C07856=1041.010,-21.005,-79.777,169.311,36.597,156.888
C07857=1041.017,-20.756,-79.792,169.314,36.598,156.888
C07858=1041.023,-20.506,-79.806,169.316,36.599,156.888
C07859=1041.030,-20.256,-79.819,169.318,36.599,156.888
C07860=1041.035,-20.007,-79.833,169.320,36.600,156.888
C07861=1041.043,-19.725,-79.849,169.322,36.601,156.888
C07862=1041.050,-19.444,-79.865,169.324,36.601,156.888
C07863=1041.057,-19.161,-79.880,169.328,36.603,156.889
C07864=1041.064,-18.880,-79.896,169.330,36.603,156.889
C07865=1041.070,-18.630,-79.910,169.332,36.604,156.889
C07866=1041.077,-18.381,-79.925,169.334,36.604,156.889
C07867=1041.083,-18.131,-79.938,169.336,36.605,156.889
C07868=1041.089,-17.881,-79.952,169.338,36.606,156.889
C07869=1041.096,-17.632,-79.966,169.340,36.606,156.889
C07870=1041.102,-17.383,-79.980,169.343,36.607,156.889
C07871=1041.109,-17.133,-79.995,169.345,36.608,156.890
C07872=1041.115,-16.884,-80.008,169.347,36.608,156.890
C07873=1041.121,-16.634,-80.023,169.349,36.609,156.890
C07874=1041.128,-16.385,-80.036,169.351,36.610,156.890
C07875=1041.134,-16.135,-80.050,169.353,36.610,156.890
C07876=1041.140,-15.886,-80.064,169.356,36.611,156.890
C07877=1041.147,-15.636,-80.078,169.358,36.611,156.890
C07878=1041.153,-15.386,-80.093,169.360,36.612,156.890
C07879=1041.160,-15.137,-80.106,169.362,36.613,156.890
C07880=1041.166,-14.887,-80.121,169.364,36.614,156.891
C07881=1041.172,-14.638,-80.135,169.366,36.615,156.891
C07882=1041.179,-14.388,-80.149,169.368,36.615,156.891
C07883=1041.184,-14.139,-80.163,169.370,36.616,156.891
C07884=1041.191,-13.889,-80.178,169.372,36.617,156.891
C07885=1041.198,-13.640,-80.193,169.374,36.617,156.891
C07886=1041.203,-13.390,-80.206,169.376,36.618,156.891
C07887=1041.210,-13.140,-80.221,169.378,36.619,156.892
C07888=1041.216,-12.891,-80.235,169.381,36.620,156.892
C07889=1041.222,-12.642,-80.250,169.383,36.620,156.892
C07890=1041.228,-12.392,-80.265,169.385,36.621,156.892
C07891=1041.235,-12.143,-80.278,169.387,36.622,156.892
C07892=1041.241,-11.893,-80.293,169.389,36.623,156.892
C07893=1041.247,-11.643,-80.307,169.391,36.623,156.892
C07894=1041.254,-11.394,-80.321,169.393,36.624,156.893
C07895=1041.260,-11.144,-80.336,169.395,36.625,156.893
C07896=1041.266,-10.895,-80.350,169.397,36.625,156.893
C07897=1041.273,-10.645,-80.364,169.399,36.627,156.893
C07898=1041.279,-10.396,-80.379,169.401,36.627,156.893
C07899=1041.285,-10.146,-80.393,169.403,36.628,156.893
C07900=1041.292,-9.897,-80.407,169.406,36.629,156.893
C07901=1041.298,-9.647,-80.422,169.408,36.629,156.893
C07902=1041.304,-9.398,-80.437,169.410,36.630,156.894
C07903=1041.311,-9.148,-80.450,169.412,36.631,156.894
C07904=1041.317,-8.899,-80.465,169.414,36.632,156.894
C07905=1041.323,-8.650,-80.480,169.416,36.632,156.894
C07906=1041.330,-8.400,-80.494,169.418,36.633,156.894
C07907=1041.336,-8.150,-80.509,169.420,36.634,156.894
C07908=1041.342,-7.901,-80.523,169.422,36.635,156.895
C07909=1041.348,-7.651,-80.538,169.424,36.636,156.895
C07910=1041.355,-7.402,-80.552,169.426,36.636,156.895
C07911=1041.361,-7.153,-80.566,169.428,36.637,156.895
C07912=1041.367,-6.903,-80.581,169.431,36.637,156.895
C07913=1041.374,-6.654,-80.596,169.433,36.639,156.895
C07914=1041.381,-6.404,-80.611,169.435,36.639,156.895
C07915=1041.386,-6.154,-80.624,169.437,36.640,156.895
C07916=1041.393,-5.905,-80.639,169.439,36.641,156.896
C07917=1041.400,-5.655,-80.654,169.441,36.641,156.896
C07918=1041.405,-5.406,-80.668,169.443,36.642,156.896
C07919=1041.412,-5.157,-80.683,169.445,36.643,156.896
C07920=1041.419,-4.907,-80.698,169.447,36.644,156.896
C07921=1041.425,-4.657,-80.712,169.449,36.644,156.896
C07922=1041.431,-4.407,-80.727,169.451,36.645,156.896
C07923=1041.437,-4.158,-80.741,169.453,36.646,156.897
C07924=1041.444,-3.909,-80.756,169.456,36.647,156.897
C07925=1041.451,-3.626,-80.772,169.459,36.648,156.897
C07926=1041.459,-3.343,-80.789,169.461,36.648,156.897
C07927=1041.466,-3.058,-80.806,169.463,36.649,156.897
C07928=1041.473,-2.775,-80.823,169.465,36.651,156.897
C07929=1041.479,-2.526,-80.837,169.467,36.651,156.898
C07930=1041.485,-2.276,-80.852,169.469,36.652,156.898
C07931=1041.491,-2.027,-80.867,169.471,36.653,156.898
C07932=1041.498,-1.777,-80.882,169.473,36.654,156.898
C07933=1041.503,-1.528,-80.897,169.476,36.655,156.898
C07934=1041.510,-1.278,-80.912,169.478,36.656,156.898
C07935=1041.516,-1.029,-80.927,169.480,36.656,156.899
C07936=1041.523,-0.779,-80.942,169.482,36.658,156.899
C07937=1041.529,-0.531,-80.957,169.484,36.658,156.899
C07938=1041.535,-0.281,-80.972,169.486,36.659,156.899
C07939=1041.541,-0.031,-80.987,169.488,36.660,156.899
C07940=1041.547,0.219,-81.002,169.489,36.661,156.899
C07941=1041.553,0.468,-81.017,169.491,36.662,156.899
C07942=1041.559,0.717,-81.032,169.493,36.663,156.900
C07943=1041.566,0.967,-81.047,169.496,36.663,156.900
C07944=1041.572,1.217,-81.062,169.498,36.664,156.900
C07945=1041.578,1.466,-81.077,169.500,36.665,156.900
C07946=1041.585,1.716,-81.092,169.502,36.666,156.900
C07947=1041.591,1.965,-81.106,169.504,36.667,156.901
C07948=1041.597,2.214,-81.121,169.506,36.668,156.901
C07949=1041.604,2.464,-81.137,169.508,36.668,156.901
C07950=1041.610,2.713,-81.152,169.510,36.670,156.901
C07951=1041.616,2.963,-81.167,169.512,36.670,156.901
C07952=1041.622,3.212,-81.181,169.514,36.671,156.901
C07953=1041.629,3.461,-81.196,169.517,36.672,156.902
C07954=1041.635,3.711,-81.211,169.518,36.673,156.902
C07955=1041.642,3.960,-81.227,169.520,36.674,156.902
C07956=1041.647,4.210,-81.242,169.522,36.675,156.902
C07957=1041.654,4.460,-81.257,169.524,36.675,156.902
C07958=1041.660,4.709,-81.272,169.526,36.677,156.902
C07959=1041.666,4.959,-81.287,169.528,36.677,156.902
C07960=1041.673,5.207,-81.303,169.530,36.678,156.903
C07961=1041.679,5.457,-81.317,169.532,36.679,156.903
C07962=1041.685,5.707,-81.332,169.534,36.680,156.903
C07963=1041.692,5.956,-81.347,169.537,36.680,156.903
C07964=1041.698,6.205,-81.363,169.539,36.682,156.903
C07965=1041.705,6.455,-81.378,169.541,36.682,156.903
C07966=1041.711,6.705,-81.393,169.542,36.683,156.904
C07967=1041.718,6.954,-81.408,169.544,36.684,156.904
C07968=1041.723,7.204,-81.424,169.546,36.685,156.904
C07969=1041.730,7.453,-81.439,169.548,36.686,156.904
C07970=1041.736,7.703,-81.454,169.550,36.687,156.904
C07971=1041.742,7.951,-81.469,169.552,36.687,156.904
C07972=1041.749,8.201,-81.484,169.554,36.689,156.905
C07973=1041.755,8.451,-81.499,169.557,36.689,156.905
C07974=1041.761,8.700,-81.514,169.559,36.690,156.905
C07975=1041.768,8.949,-81.530,169.561,36.691,156.905
C07976=1041.775,9.199,-81.545,169.563,36.692,156.905
C07977=1041.780,9.449,-81.560,169.564,36.692,156.905
C07978=1041.787,9.698,-81.576,169.566,36.694,156.906
C07979=1041.793,9.948,-81.591,169.568,36.694,156.906
C07980=1041.800,10.197,-81.607,169.570,36.695,156.906
C07981=1041.806,10.446,-81.622,169.572,36.696,156.906
C07982=1041.813,10.696,-81.636,169.574,36.697,156.906
C07983=1041.819,10.945,-81.652,169.576,36.698,156.906
C07984=1041.826,11.195,-81.667,169.579,36.699,156.906
C07985=1041.833,11.444,-81.683,169.581,36.699,156.907
C07986=1041.838,11.694,-81.698,169.583,36.700,156.907
C07987=1041.845,11.943,-81.713,169.585,36.701,156.907
C07988=1041.851,12.192,-81.729,169.586,36.702,156.907
C07989=1041.859,12.478,-81.747,169.589,36.703,156.907
C07990=1041.866,12.764,-81.764,169.591,36.704,156.907
C07991=1041.874,13.049,-81.781,169.593,36.705,156.908
C07992=1041.881,13.334,-81.799,169.595,36.706,156.908
C07993=1041.887,13.584,-81.814,169.598,36.707,156.908
C07994=1041.893,13.833,-81.830,169.600,36.708,156.908
C07995=1041.900,14.083,-81.845,169.602,36.708,156.908
C07996=1041.906,14.332,-81.861,169.604,36.709,156.908
C07997=1041.913,14.581,-81.876,169.606,36.710,156.909
C07998=1041.919,14.831,-81.892,169.607,36.711,156.909
C07999=1041.925,15.080,-81.908,169.609,36.712,156.909
C08000=1041.931,15.330,-81.923,169.611,36.713,156.909
C08001=1041.938,15.579,-81.939,169.613,36.714,156.909
C08002=1041.944,15.828,-81.954,169.616,36.715,156.910
C08003=1041.950,16.078,-81.970,169.618,36.716,156.910
C08004=1041.957,16.327,-81.986,169.620,36.717,156.910
C08005=1041.962,16.577,-82.001,169.621,36.718,156.910
C08006=1041.969,16.826,-82.017,169.623,36.719,156.910
C08007=1041.976,17.076,-82.032,169.625,36.720,156.910
C08008=1041.982,17.325,-82.048,169.627,36.721,156.911
C08009=1041.989,17.575,-82.064,169.629,36.721,156.911
C08010=1041.994,17.824,-82.080,169.631,36.723,156.911
C08011=1042.001,18.074,-82.095,169.634,36.723,156.911
C08012=1042.008,18.323,-82.111,169.635,36.725,156.911
C08013=1042.013,18.573,-82.126,169.637,36.725,156.911
C08014=1042.020,18.822,-82.142,169.639,36.726,156.912
C08015=1042.026,19.071,-82.158,169.641,36.727,156.912
C08016=1042.032,19.321,-82.173,169.643,36.728,156.912
C08017=1042.039,19.570,-82.189,169.645,36.729,156.912
C08018=1042.045,19.819,-82.205,169.647,36.730,156.912
C08019=1042.052,20.069,-82.221,169.648,36.731,156.913
C08020=1042.058,20.319,-82.237,169.651,36.732,156.913
C08021=1042.065,20.568,-82.252,169.653,36.733,156.913
C08022=1042.071,20.817,-82.269,169.655,36.734,156.913
C08023=1042.077,21.066,-82.284,169.657,36.735,156.913
C08024=1042.083,21.316,-82.300,169.659,36.736,156.913
C08025=1042.090,21.565,-82.316,169.660,36.737,156.914
C08026=1042.096,21.814,-82.332,169.662,36.738,156.914
C08027=1042.102,22.064,-82.348,169.664,36.738,156.914
C08028=1042.109,22.314,-82.364,169.666,36.740,156.914
C08029=1042.115,22.563,-82.380,169.669,36.740,156.914
C08030=1042.121,22.813,-82.395,169.671,36.742,156.915
C08031=1042.127,23.062,-82.412,169.672,36.742,156.915
C08032=1042.134,23.311,-82.427,169.674,36.743,156.915
C08033=1042.140,23.560,-82.444,169.676,36.744,156.915
C08034=1042.147,23.809,-82.459,169.678,36.745,156.915
C08035=1042.153,24.060,-82.475,169.680,36.746,156.915
C08036=1042.159,24.309,-82.491,169.681,36.747,156.916
C08037=1042.165,24.558,-82.507,169.684,36.748,156.916
C08038=1042.171,24.808,-82.523,169.686,36.749,156.916
C08039=1042.178,25.057,-82.539,169.688,36.750,156.916
C08040=1042.185,25.307,-82.556,169.690,36.751,156.916
C08041=1042.191,25.556,-82.571,169.692,36.752,156.917
C08042=1042.197,25.805,-82.587,169.693,36.753,156.917
C08043=1042.204,26.054,-82.603,169.695,36.754,156.917
C08044=1042.210,26.304,-82.619,169.697,36.755,156.917
C08045=1042.216,26.554,-82.636,169.699,36.756,156.917
C08046=1042.223,26.803,-82.651,169.702,36.757,156.917
C08047=1042.229,27.053,-82.667,169.704,36.758,156.918
C08048=1042.235,27.302,-82.683,169.705,36.759,156.918
C08049=1042.241,27.551,-82.699,169.707,36.760,156.918
C08050=1042.248,27.801,-82.716,169.709,36.760,156.918
C08051=1042.255,28.050,-82.731,169.711,36.762,156.918
C08052=1042.261,28.299,-82.748,169.713,36.763,156.919
C08053=1042.268,28.586,-82.766,169.715,36.764,156.919
C08054=1042.275,28.872,-82.786,169.718,36.765,156.919
C08055=1042.282,29.160,-82.804,169.720,36.766,156.919
C08056=1042.290,29.446,-82.822,169.722,36.767,156.919
C08057=1042.296,29.695,-82.839,169.724,36.769,156.920
C08058=1042.302,29.945,-82.855,169.725,36.769,156.920
C08059=1042.308,30.194,-82.871,169.727,36.770,156.920
C08060=1042.315,30.444,-82.887,169.729,36.772,156.920
C08061=1042.321,30.693,-82.904,169.731,36.772,156.920
C08062=1042.327,30.942,-82.921,169.734,36.774,156.921
C08063=1042.333,31.191,-82.937,169.735,36.774,156.921
C08064=1042.340,31.441,-82.953,169.737,36.775,156.921
C08065=1042.346,31.690,-82.969,169.739,36.777,156.921
C08066=1042.352,31.940,-82.985,169.741,36.777,156.921
C08067=1042.358,32.189,-83.002,169.743,36.779,156.922
C08068=1042.365,32.438,-83.019,169.744,36.780,156.922
C08069=1042.372,32.688,-83.035,169.746,36.780,156.922
C08070=1042.378,32.937,-83.051,169.749,36.782,156.922
C08071=1042.384,33.187,-83.067,169.751,36.782,156.922
C08072=1042.390,33.436,-83.084,169.753,36.784,156.923
C08073=1042.396,33.686,-83.100,169.754,36.785,156.923
C08074=1042.402,33.934,-83.117,169.756,36.785,156.923
C08075=1042.410,34.184,-83.133,169.758,36.787,156.923
C08076=1042.416,34.433,-83.149,169.760,36.787,156.923
C08077=1042.422,34.683,-83.165,169.762,36.789,156.924
C08078=1042.428,34.933,-83.182,169.764,36.790,156.924
C08079=1042.434,35.182,-83.199,169.766,36.790,156.924
C08080=1042.441,35.431,-83.215,169.768,36.792,156.924
C08081=1042.448,35.681,-83.231,169.770,36.792,156.924
C08082=1042.454,35.930,-83.248,169.771,36.794,156.924
C08083=1042.460,36.179,-83.265,169.773,36.795,156.925
C08084=1042.466,36.429,-83.281,169.775,36.795,156.925
C08085=1042.472,36.678,-83.297,169.777,36.797,156.925
C08086=1042.479,36.927,-83.314,169.779,36.797,156.925
C08087=1042.486,37.177,-83.330,169.781,36.799,156.925
C08088=1042.492,37.426,-83.347,169.783,36.800,156.926
C08089=1042.498,37.675,-83.363,169.785,36.800,156.926
C08090=1042.505,37.925,-83.380,169.787,36.802,156.926
C08091=1042.511,38.174,-83.397,169.788,36.803,156.926
C08092=1042.517,38.423,-83.414,169.790,36.804,156.926
C08093=1042.523,38.673,-83.430,169.792,36.805,156.927
C08094=1042.529,38.922,-83.446,169.795,36.806,156.927
C08095=1042.536,39.172,-83.464,169.797,36.807,156.927
C08096=1042.542,39.421,-83.480,169.798,36.808,156.927
C08097=1042.548,39.670,-83.496,169.800,36.809,156.927
C08098=1042.554,39.920,-83.514,169.802,36.810,156.928
C08099=1042.560,40.169,-83.530,169.804,36.811,156.928
C08100=1042.566,40.418,-83.547,169.805,36.812,156.928
C08101=1042.573,40.668,-83.564,169.807,36.814,156.928
C08102=1042.579,40.917,-83.581,169.810,36.814,156.928
C08103=1042.586,41.167,-83.598,169.812,36.815,156.929
C08104=1042.592,41.416,-83.615,169.813,36.817,156.929
C08105=1042.598,41.665,-83.631,169.815,36.818,156.929
C08106=1042.605,41.915,-83.647,169.817,36.819,156.929
C08107=1042.611,42.164,-83.664,169.819,36.820,156.930
C08108=1042.617,42.414,-83.681,169.820,36.821,156.930
C08109=1042.624,42.663,-83.698,169.822,36.822,156.930
C08110=1042.630,42.912,-83.714,169.825,36.823,156.930
C08111=1042.636,43.161,-83.732,169.827,36.824,156.930
C08112=1042.643,43.410,-83.749,169.828,36.825,156.930
C08113=1042.649,43.660,-83.766,169.830,36.826,156.931
C08114=1042.655,43.909,-83.783,169.832,36.827,156.931
C08115=1042.661,44.159,-83.799,169.834,36.829,156.931
C08116=1042.667,44.408,-83.817,169.835,36.830,156.931
C08117=1042.674,44.695,-83.836,169.838,36.831,156.932
C08118=1042.681,44.980,-83.856,169.840,36.832,156.932
C08119=1042.688,45.268,-83.875,169.842,36.834,156.932
C08120=1042.695,45.554,-83.894,169.844,36.835,156.932
C08121=1042.701,45.804,-83.912,169.846,36.836,156.933
C08122=1042.708,46.053,-83.929,169.848,36.837,156.933
C08123=1042.713,46.302,-83.946,169.850,36.838,156.933
C08124=1042.720,46.552,-83.963,169.852,36.839,156.933
C08125=1042.726,46.801,-83.981,169.854,36.840,156.933
C08126=1042.732,47.051,-83.997,169.856,36.842,156.934
C08127=1042.739,47.299,-84.014,169.857,36.843,156.934
C08128=1042.745,47.549,-84.032,169.859,36.844,156.934
C08129=1042.751,47.798,-84.048,169.861,36.845,156.934
C08130=1042.758,48.048,-84.066,169.864,36.846,156.935
C08131=1042.763,48.297,-84.083,169.865,36.847,156.935
C08132=1042.770,48.546,-84.101,169.867,36.849,156.935
C08133=1042.776,48.796,-84.117,169.869,36.850,156.935
C08134=1042.781,49.045,-84.134,169.870,36.850,156.935
C08135=1042.788,49.294,-84.152,169.872,36.852,156.936
C08136=1042.794,49.544,-84.168,169.874,36.853,156.936
C08137=1042.800,49.793,-84.186,169.877,36.854,156.936
C08138=1042.807,50.042,-84.203,169.878,36.855,156.936
C08139=1042.813,50.291,-84.220,169.880,36.856,156.937
C08140=1042.819,50.540,-84.238,169.882,36.857,156.937
C08141=1042.826,50.791,-84.254,169.884,36.859,156.937
C08142=1042.831,51.040,-84.272,169.885,36.860,156.937
C08143=1042.838,51.289,-84.289,169.887,36.860,156.937
C08144=1042.844,51.538,-84.306,169.889,36.862,156.938
C08145=1042.850,51.787,-84.324,169.891,36.863,156.938
C08146=1042.857,52.038,-84.341,169.893,36.864,156.938
C08147=1042.863,52.286,-84.358,169.895,36.865,156.938
C08148=1042.869,52.536,-84.376,169.897,36.866,156.938
C08149=1042.875,52.785,-84.393,169.898,36.867,156.939
C08150=1042.882,53.034,-84.410,169.900,36.869,156.939
C08151=1042.888,53.283,-84.428,169.902,36.870,156.939
C08152=1042.894,53.533,-84.444,169.905,36.870,156.939
C08153=1042.900,53.782,-84.462,169.906,36.872,156.940
C08154=1042.907,54.032,-84.479,169.908,36.873,156.940
C08155=1042.914,54.281,-84.496,169.910,36.874,156.940
C08156=1042.919,54.530,-84.514,169.911,36.875,156.940
C08157=1042.926,54.780,-84.531,169.913,36.876,156.940
C08158=1042.932,55.028,-84.548,169.915,36.877,156.941
C08159=1042.938,55.278,-84.566,169.918,36.878,156.941
C08160=1042.945,55.527,-84.584,169.919,36.879,156.941
C08161=1042.951,55.777,-84.601,169.921,36.880,156.941
C08162=1042.958,56.026,-84.619,169.923,36.882,156.941
C08163=1042.964,56.275,-84.635,169.925,36.883,156.942
C08164=1042.970,56.525,-84.653,169.926,36.883,156.942
C08165=1042.977,56.774,-84.670,169.928,36.885,156.942
C08166=1042.983,57.023,-84.687,169.931,36.886,156.942
C08167=1042.989,57.273,-84.705,169.933,36.887,156.943
C08168=1042.996,57.522,-84.722,169.934,36.888,156.943
C08169=1043.001,57.771,-84.740,169.936,36.889,156.943
C08170=1043.008,58.021,-84.757,169.938,36.890,156.943
C08171=1043.014,58.270,-84.774,169.939,36.892,156.943
C08172=1043.021,58.519,-84.792,169.941,36.892,156.944
C08173=1043.027,58.769,-84.809,169.943,36.893,156.944
C08174=1043.033,59.018,-84.827,169.946,36.895,156.944
C08175=1043.040,59.267,-84.844,169.947,36.896,156.944
C08176=1043.047,59.517,-84.862,169.949,36.897,156.944
C08177=1043.052,59.765,-84.880,169.951,36.898,156.945
C08178=1043.059,60.014,-84.897,169.953,36.899,156.945
C08179=1043.065,60.264,-84.915,169.954,36.900,156.945
C08180=1043.072,60.514,-84.933,169.956,36.901,156.945
C08181=1043.079,60.800,-84.953,169.959,36.902,156.945
C08182=1043.087,61.086,-84.973,169.961,36.903,156.946
C08183=1043.094,61.372,-84.993,169.963,36.905,156.946
C08184=1043.101,61.659,-85.013,169.965,36.906,156.946
C08185=1043.108,61.908,-85.030,169.967,36.907,156.946
C08186=1043.114,62.157,-85.048,169.969,36.908,156.947
C08187=1043.121,62.407,-85.065,169.970,36.909,156.947
C08188=1043.127,62.656,-85.083,169.973,36.910,156.947
C08189=1043.133,62.905,-85.101,169.975,36.911,156.947
C08190=1043.140,63.154,-85.118,169.977,36.912,156.947
C08191=1043.146,63.404,-85.136,169.978,36.913,156.948
C08192=1043.153,63.653,-85.154,169.980,36.914,156.948
C08193=1043.159,63.902,-85.171,169.982,36.915,156.948
C08194=1043.166,64.152,-85.188,169.984,36.916,156.948
C08195=1043.172,64.401,-85.207,169.986,36.918,156.949
C08196=1043.178,64.651,-85.225,169.988,36.919,156.949
C08197=1043.184,64.899,-85.242,169.990,36.920,156.949
C08198=1043.190,65.149,-85.260,169.991,36.921,156.949
C08199=1043.197,65.398,-85.279,169.993,36.922,156.949
C08200=1043.202,65.647,-85.296,169.995,36.923,156.950
C08201=1043.209,65.897,-85.314,169.996,36.924,156.950
C08202=1043.216,66.146,-85.332,169.999,36.926,156.950
C08203=1043.222,66.395,-85.350,170.001,36.927,156.950
C08204=1043.228,66.644,-85.367,170.003,36.928,156.951
C08205=1043.234,66.894,-85.385,170.004,36.929,156.951
C08206=1043.241,67.143,-85.404,170.006,36.930,156.951
C08207=1043.247,67.392,-85.421,170.008,36.931,156.951
C08208=1043.253,67.641,-85.439,170.010,36.932,156.951
C08209=1043.259,67.891,-85.457,170.012,36.934,156.952
C08210=1043.265,68.140,-85.475,170.014,36.935,156.952
C08211=1043.273,68.389,-85.493,170.016,36.936,156.952
C08212=1043.278,68.638,-85.511,170.017,36.937,156.952
C08213=1043.284,68.888,-85.529,170.019,36.938,156.953
C08214=1043.291,69.137,-85.547,170.021,36.939,156.953
C08215=1043.298,69.387,-85.565,170.023,36.941,156.953
C08216=1043.304,69.636,-85.583,170.025,36.942,156.953
C08217=1043.310,69.885,-85.601,170.027,36.943,156.953
C08218=1043.316,70.134,-85.619,170.029,36.944,156.954
C08219=1043.322,70.384,-85.637,170.030,36.945,156.954
C08220=1043.328,70.633,-85.655,170.032,36.946,156.954
C08221=1043.334,70.882,-85.674,170.034,36.947,156.954
C08222=1043.340,71.131,-85.692,170.036,36.949,156.955
C08223=1043.347,71.380,-85.710,170.038,36.950,156.955
C08224=1043.353,71.630,-85.728,170.040,36.951,156.955
C08225=1043.360,71.879,-85.746,170.041,36.952,156.955
C08226=1043.365,72.128,-85.764,170.043,36.954,156.956
C08227=1043.372,72.377,-85.782,170.045,36.955,156.956
C08228=1043.378,72.627,-85.800,170.048,36.956,156.956
C08229=1043.384,72.876,-85.819,170.049,36.957,156.956
C08230=1043.390,73.126,-85.837,170.051,36.958,156.956
C08231=1043.396,73.374,-85.855,170.053,36.959,156.957
C08232=1043.402,73.624,-85.873,170.054,36.960,156.957
C08233=1043.409,73.873,-85.892,170.056,36.962,156.957
C08234=1043.415,74.123,-85.910,170.058,36.963,156.957
C08235=1043.422,74.372,-85.928,170.060,36.964,156.958
C08236=1043.429,74.621,-85.947,170.062,36.965,156.958
C08237=1043.435,74.871,-85.964,170.064,36.967,156.958
C08238=1043.440,75.119,-85.983,170.066,36.967,156.958
C08239=1043.447,75.369,-86.001,170.067,36.968,156.958
C08240=1043.453,75.618,-86.019,170.069,36.970,156.959
C08241=1043.459,75.867,-86.038,170.072,36.971,156.959
C08242=1043.466,76.117,-86.056,170.073,36.972,156.959
C08243=1043.472,76.366,-86.075,170.075,36.973,156.959
C08244=1043.478,76.616,-86.092,170.077,36.975,156.960
C08245=1043.485,76.901,-86.113,170.079,36.976,156.960
C08246=1043.493,77.187,-86.135,170.081,36.977,156.960
C08247=1043.500,77.473,-86.155,170.083,36.978,156.960
C08248=1043.507,77.759,-86.177,170.086,36.979,156.961
C08249=1043.513,78.009,-86.195,170.087,36.981,156.961
C08250=1043.519,78.258,-86.214,170.089,36.982,156.961
C08251=1043.526,78.507,-86.232,170.091,36.983,156.961
C08252=1043.532,78.756,-86.251,170.092,36.984,156.962
C08253=1043.538,79.006,-86.269,170.094,36.986,156.962
C08254=1043.544,79.254,-86.288,170.097,36.987,156.962
C08255=1043.550,79.504,-86.306,170.099,36.988,156.962
C08256=1043.556,79.753,-86.325,170.100,36.989,156.963
C08257=1043.563,80.002,-86.343,170.102,36.991,156.963
C08258=1043.568,80.252,-86.362,170.104,36.992,156.963
C08259=1043.575,80.501,-86.381,170.105,36.993,156.963
C08260=1043.581,80.750,-86.400,170.108,36.994,156.964
C08261=1043.587,80.999,-86.418,170.110,36.996,156.964
C08262=1043.594,81.249,-86.436,170.111,36.997,156.964
C08263=1043.599,81.498,-86.455,170.113,36.998,156.964
C08264=1043.605,81.747,-86.474,170.115,36.999,156.965
C08265=1043.612,81.996,-86.492,170.116,37.000,156.965
C08266=1043.618,82.245,-86.511,170.119,37.002,156.965
C08267=1043.624,82.494,-86.530,170.121,37.003,156.965
C08268=1043.630,82.744,-86.549,170.123,37.004,156.966
C08269=1043.636,82.993,-86.567,170.124,37.005,156.966
C08270=1043.643,83.242,-86.585,170.126,37.007,156.966
C08271=1043.649,83.492,-86.604,170.128,37.008,156.966
C08272=1043.655,83.741,-86.623,170.130,37.009,156.967
C08273=1043.661,83.990,-86.642,170.132,37.010,156.967
C08274=1043.668,84.239,-86.661,170.134,37.012,156.967
C08275=1043.674,84.488,-86.679,170.135,37.013,156.967
C08276=1043.680,84.738,-86.698,170.137,37.014,156.968
C08277=1043.687,84.987,-86.717,170.139,37.015,156.968
C08278=1043.693,85.236,-86.736,170.141,37.016,156.968
C08279=1043.699,85.485,-86.754,170.143,37.017,156.968
C08280=1043.705,85.734,-86.773,170.145,37.018,156.968
C08281=1043.712,85.983,-86.792,170.147,37.020,156.969
C08282=1043.717,86.233,-86.810,170.148,37.021,156.969
C08283=1043.724,86.483,-86.829,170.150,37.022,156.969
C08284=1043.730,86.732,-86.848,170.152,37.023,156.969
C08285=1043.736,86.981,-86.866,170.154,37.025,156.970
C08286=1043.742,87.230,-86.885,170.156,37.026,156.970
C08287=1043.749,87.479,-86.904,170.158,37.027,156.970
C08288=1043.755,87.729,-86.923,170.160,37.028,156.970
C08289=1043.762,87.977,-86.942,170.161,37.029,156.971
C08290=1043.767,88.226,-86.961,170.163,37.031,156.971
C08291=1043.774,88.476,-86.980,170.166,37.032,156.971
C08292=1043.780,88.725,-86.999,170.167,37.033,156.971
C08293=1043.787,88.974,-87.017,170.169,37.034,156.971
C08294=1043.792,89.223,-87.037,170.171,37.035,156.972
C08295=1043.799,89.472,-87.055,170.173,37.036,156.972
C08296=1043.805,89.722,-87.074,170.174,37.037,156.972
C08297=1043.812,89.971,-87.092,170.177,37.039,156.972
C08298=1043.818,90.221,-87.112,170.179,37.040,156.973
C08299=1043.824,90.470,-87.131,170.181,37.041,156.973
C08300=1043.830,90.719,-87.150,170.182,37.042,156.973
C08301=1043.837,90.968,-87.169,170.184,37.044,156.973
C08302=1043.843,91.217,-87.189,170.186,37.045,156.974
C08303=1043.849,91.466,-87.207,170.188,37.046,156.974
C08304=1043.855,91.716,-87.226,170.190,37.047,156.974
C08305=1043.861,91.965,-87.245,170.192,37.049,156.974
C08306=1043.867,92.214,-87.264,170.193,37.050,156.975
C08307=1043.873,92.463,-87.284,170.195,37.052,156.975
C08308=1043.879,92.712,-87.303,170.197,37.053,156.975
C08309=1043.886,92.999,-87.325,170.200,37.054,156.976
C08310=1043.894,93.284,-87.347,170.202,37.055,156.976
C08311=1043.901,93.571,-87.369,170.204,37.057,156.976
C08312=1043.908,93.856,-87.391,170.206,37.058,156.976
C08313=1043.913,94.105,-87.410,170.207,37.060,156.977
C08314=1043.920,94.355,-87.429,170.210,37.061,156.977
C08315=1043.926,94.604,-87.448,170.212,37.062,156.977
C08316=1043.933,94.853,-87.467,170.213,37.063,156.977
C08317=1043.939,95.102,-87.487,170.215,37.064,156.978
C08318=1043.945,95.351,-87.505,170.217,37.066,156.978
C08319=1043.951,95.600,-87.525,170.219,37.067,156.978
C08320=1043.957,95.850,-87.545,170.221,37.068,156.978
C08321=1043.963,96.099,-87.563,170.223,37.069,156.979
C08322=1043.969,96.348,-87.583,170.225,37.071,156.979
C08323=1043.976,96.597,-87.602,170.226,37.072,156.979
C08324=1043.982,96.847,-87.621,170.228,37.073,156.979
C08325=1043.989,97.095,-87.641,170.230,37.074,156.980
C08326=1043.994,97.345,-87.660,170.233,37.076,156.980
C08327=1044.001,97.594,-87.679,170.234,37.077,156.980
C08328=1044.007,97.843,-87.699,170.236,37.078,156.980
C08329=1044.014,98.093,-87.718,170.238,37.079,156.981
C08330=1044.020,98.341,-87.738,170.239,37.080,156.981
C08331=1044.025,98.591,-87.757,170.241,37.082,156.981
C08332=1044.032,98.840,-87.775,170.244,37.083,156.981
C08333=1044.038,99.089,-87.795,170.246,37.084,156.982
C08334=1044.044,99.338,-87.814,170.247,37.085,156.982
C08335=1044.051,99.587,-87.834,170.249,37.087,156.982
C08336=1044.057,99.836,-87.853,170.251,37.088,156.982
C08337=1044.063,100.086,-87.872,170.253,37.089,156.983
C08338=1044.070,100.334,-87.892,170.255,37.090,156.983
C08339=1044.075,100.584,-87.911,170.257,37.091,156.983
C08340=1044.082,100.833,-87.931,170.259,37.093,156.983
C08341=1044.088,101.083,-87.950,170.260,37.095,156.984
C08342=1044.094,101.332,-87.970,170.262,37.096,156.984
C08343=1044.100,101.581,-87.989,170.264,37.097,156.984
C08344=1044.106,101.830,-88.009,170.267,37.098,156.984
C08345=1044.113,102.079,-88.029,170.268,37.099,156.985
C08346=1044.118,102.328,-88.049,170.270,37.101,156.985
C08347=1044.124,102.577,-88.069,170.272,37.102,156.985
C08348=1044.131,102.826,-88.087,170.273,37.104,156.986
C08349=1044.137,103.075,-88.107,170.276,37.105,156.986
C08350=1044.142,103.325,-88.126,170.278,37.106,156.986
C08351=1044.149,103.574,-88.147,170.280,37.107,156.986
C08352=1044.155,103.823,-88.167,170.281,37.109,156.987
C08353=1044.161,104.072,-88.186,170.283,37.110,156.987
C08354=1044.167,104.321,-88.205,170.285,37.111,156.987
C08355=1044.174,104.570,-88.226,170.287,37.112,156.987
C08356=1044.180,104.820,-88.245,170.289,37.114,156.988
C08357=1044.186,105.069,-88.265,170.291,37.115,156.988
C08358=1044.191,105.318,-88.284,170.293,37.117,156.988
C08359=1044.199,105.567,-88.304,170.294,37.118,156.988
C08360=1044.205,105.816,-88.324,170.297,37.119,156.989
C08361=1044.210,106.066,-88.343,170.299,37.120,156.989
C08362=1044.216,106.314,-88.363,170.301,37.121,156.989
C08363=1044.223,106.564,-88.383,170.302,37.123,156.989
C08364=1044.229,106.813,-88.403,170.304,37.124,156.990
C08365=1044.235,107.062,-88.422,170.306,37.125,156.990
C08366=1044.241,107.311,-88.442,170.308,37.126,156.990
C08367=1044.248,107.560,-88.462,170.310,37.128,156.990
C08368=1044.254,107.810,-88.481,170.312,37.129,156.991
C08369=1044.260,108.058,-88.501,170.314,37.131,156.991
C08370=1044.266,108.308,-88.522,170.315,37.132,156.991
C08371=1044.272,108.557,-88.542,170.317,37.133,156.991
C08372=1044.279,108.806,-88.560,170.320,37.134,156.992
C08373=1044.285,109.092,-88.583,170.322,37.136,156.992
C08374=1044.293,109.379,-88.607,170.324,37.137,156.992
C08375=1044.300,109.664,-88.630,170.326,37.139,156.993
C08376=1044.307,109.950,-88.653,170.328,37.140,156.993
C08377=1044.313,110.199,-88.672,170.331,37.141,156.993
C08378=1044.320,110.448,-88.692,170.332,37.142,156.993
C08379=1044.326,110.697,-88.711,170.334,37.144,156.994
C08380=1044.332,110.946,-88.731,170.336,37.145,156.994
C08381=1044.339,111.195,-88.752,170.338,37.147,156.994
C08382=1044.345,111.444,-88.772,170.340,37.148,156.994
C08383=1044.350,111.694,-88.791,170.342,37.149,156.995
C08384=1044.357,111.943,-88.811,170.344,37.150,156.995
C08385=1044.363,112.192,-88.831,170.346,37.151,156.995
C08386=1044.369,112.441,-88.851,170.347,37.153,156.996
C08387=1044.376,112.690,-88.872,170.349,37.155,156.996
C08388=1044.382,112.939,-88.892,170.352,37.156,156.996
C08389=1044.388,113.188,-88.911,170.354,37.157,156.996
C08390=1044.394,113.438,-88.932,170.355,37.158,156.997
C08391=1044.399,113.687,-88.952,170.357,37.159,156.997
C08392=1044.405,113.935,-88.972,170.359,37.161,156.997
C08393=1044.412,114.185,-88.993,170.362,37.162,156.997
C08394=1044.418,114.434,-89.013,170.363,37.164,156.998
C08395=1044.423,114.683,-89.033,170.365,37.165,156.998
C08396=1044.430,114.932,-89.053,170.367,37.167,156.998
C08397=1044.436,115.181,-89.073,170.369,37.168,156.999
C08398=1044.442,115.430,-89.093,170.371,37.169,156.999
C08399=1044.448,115.680,-89.114,170.373,37.170,156.999
C08400=1044.454,115.929,-89.134,170.375,37.172,156.999
C08401=1044.460,116.177,-89.154,170.376,37.173,157.000
C08402=1044.466,116.427,-89.175,170.378,37.175,157.000
C08403=1044.472,116.676,-89.195,170.380,37.176,157.000
C08404=1044.478,116.925,-89.215,170.383,37.178,157.001
C08405=1044.484,117.174,-89.236,170.384,37.179,157.001
C08406=1044.490,117.423,-89.257,170.386,37.180,157.001
C08407=1044.496,117.672,-89.277,170.388,37.181,157.001
C08408=1044.502,117.921,-89.297,170.391,37.183,157.002
C08409=1044.508,118.170,-89.317,170.392,37.184,157.002
C08410=1044.514,118.420,-89.338,170.394,37.186,157.002
C08411=1044.520,118.669,-89.358,170.396,37.187,157.002
C08412=1044.527,118.918,-89.378,170.398,37.189,157.003
C08413=1044.532,119.167,-89.399,170.399,37.190,157.003
C08414=1044.538,119.416,-89.419,170.402,37.191,157.003
C08415=1044.545,119.665,-89.440,170.404,37.192,157.004
C08416=1044.550,119.914,-89.460,170.406,37.194,157.004
C08417=1044.557,120.164,-89.481,170.407,37.195,157.004
C08418=1044.563,120.412,-89.501,170.409,37.197,157.004
C08419=1044.570,120.661,-89.522,170.412,37.198,157.005
C08420=1044.575,120.911,-89.542,170.414,37.200,157.005
C08421=1044.581,121.159,-89.562,170.416,37.201,157.005
C08422=1044.587,121.409,-89.582,170.417,37.202,157.006
C08423=1044.593,121.657,-89.604,170.419,37.203,157.006
C08424=1044.600,121.907,-89.624,170.422,37.204,157.006
C08425=1044.606,122.156,-89.644,170.424,37.206,157.006
C08426=1044.611,122.406,-89.665,170.425,37.208,157.007
C08427=1044.618,122.654,-89.686,170.427,37.209,157.007
C08428=1044.624,122.903,-89.706,170.429,37.210,157.007
C08429=1044.630,123.152,-89.726,170.432,37.212,157.008
C08430=1044.637,123.401,-89.747,170.434,37.213,157.008
C08431=1044.643,123.650,-89.767,170.435,37.214,157.008
C08432=1044.648,123.900,-89.788,170.437,37.215,157.008
C08433=1044.655,124.148,-89.809,170.439,37.217,157.009
C08434=1044.661,124.398,-89.829,170.442,37.218,157.009
C08435=1044.667,124.647,-89.850,170.444,37.220,157.009
C08436=1044.673,124.896,-89.871,170.445,37.221,157.009
C08437=1044.680,125.182,-89.894,170.447,37.223,157.010
C08438=1044.688,125.468,-89.918,170.449,37.224,157.010
C08439=1044.695,125.753,-89.942,170.453,37.226,157.010
C08440=1044.702,126.039,-89.965,170.455,37.227,157.011
C08441=1044.708,126.288,-89.986,170.456,37.228,157.011
C08442=1044.714,126.537,-90.006,170.458,37.230,157.011
C08443=1044.720,126.786,-90.027,170.460,37.231,157.012
C08444=1044.726,127.036,-90.048,170.463,37.232,157.012
C08445=1044.733,127.284,-90.069,170.465,37.234,157.012
C08446=1044.739,127.534,-90.089,170.466,37.235,157.012
C08447=1044.745,127.782,-90.110,170.468,37.237,157.013
C08448=1044.751,128.032,-90.131,170.470,37.238,157.013
C08449=1044.757,128.280,-90.151,170.473,37.239,157.013
C08450=1044.764,128.530,-90.172,170.475,37.240,157.013
C08451=1044.770,128.779,-90.193,170.477,37.242,157.014
C08452=1044.776,129.028,-90.214,170.478,37.243,157.014
C08453=1044.782,129.277,-90.234,170.480,37.245,157.014
C08454=1044.789,129.526,-90.255,170.483,37.246,157.015
C08455=1044.794,129.775,-90.276,170.485,37.247,157.015
C08456=1044.801,130.024,-90.297,170.487,37.248,157.015
C08457=1044.807,130.273,-90.317,170.489,37.250,157.015
C08458=1044.814,130.522,-90.338,170.490,37.251,157.016
C08459=1044.820,130.772,-90.359,170.493,37.252,157.016
C08460=1044.826,131.020,-90.380,170.495,37.254,157.016
C08461=1044.833,131.269,-90.401,170.497,37.255,157.016
C08462=1044.838,131.519,-90.422,170.499,37.257,157.017
C08463=1044.845,131.767,-90.443,170.500,37.258,157.017
C08464=1044.851,132.017,-90.464,170.502,37.259,157.017
C08465=1044.857,132.266,-90.485,170.505,37.261,157.018
C08466=1044.863,132.514,-90.506,170.507,37.262,157.018
C08467=1044.869,132.764,-90.527,170.509,37.263,157.018
C08468=1044.874,133.013,-90.548,170.511,37.265,157.019
C08469=1044.881,133.261,-90.569,170.513,37.266,157.019
C08470=1044.887,133.511,-90.590,170.515,37.268,157.019
C08471=1044.893,133.760,-90.611,170.517,37.269,157.019
C08472=1044.900,134.009,-90.632,170.519,37.271,157.020
C08473=1044.906,134.258,-90.654,170.521,37.272,157.020
C08474=1044.911,134.507,-90.674,170.523,37.274,157.020
C08475=1044.918,134.756,-90.696,170.525,37.275,157.021
C08476=1044.924,135.004,-90.717,170.527,37.276,157.021
C08477=1044.929,135.254,-90.738,170.529,37.278,157.021
C08478=1044.936,135.503,-90.759,170.531,37.279,157.021
C08479=1044.942,135.752,-90.780,170.534,37.280,157.022
C08480=1044.948,136.001,-90.802,170.536,37.282,157.022
C08481=1044.955,136.250,-90.823,170.537,37.283,157.022
C08482=1044.961,136.500,-90.844,170.539,37.285,157.023
C08483=1044.966,136.748,-90.865,170.541,37.286,157.023
C08484=1044.973,136.997,-90.887,170.544,37.288,157.023
C08485=1044.979,137.246,-90.908,170.546,37.289,157.023
C08486=1044.985,137.495,-90.929,170.548,37.291,157.024
C08487=1044.991,137.745,-90.950,170.549,37.292,157.024
C08488=1044.997,137.994,-90.971,170.551,37.293,157.024
C08489=1045.003,138.242,-90.992,170.554,37.295,157.025
C08490=1045.009,138.491,-91.014,170.556,37.296,157.025
C08491=1045.016,138.740,-91.035,170.558,37.298,157.025
C08492=1045.022,138.990,-91.057,170.560,37.299,157.026
C08493=1045.028,139.238,-91.078,170.563,37.300,157.026
C08494=1045.034,139.487,-91.099,170.564,37.302,157.026
C08495=1045.040,139.737,-91.120,170.566,37.303,157.027
C08496=1045.046,139.986,-91.142,170.568,37.305,157.027
C08497=1045.052,140.234,-91.163,170.570,37.306,157.027
C08498=1045.058,140.484,-91.185,170.573,37.308,157.027
C08499=1045.064,140.733,-91.206,170.575,37.309,157.028
C08500=1045.070,140.981,-91.228,170.577,37.311,157.028
C08501=1045.078,141.267,-91.252,170.579,37.312,157.028
C08502=1045.084,141.553,-91.277,170.582,37.314,157.029
C08503=1045.091,141.838,-91.302,170.584,37.316,157.029
C08504=1045.098,142.123,-91.327,170.586,37.317,157.029
C08505=1045.104,142.373,-91.349,170.588,37.319,157.030
C08506=1045.111,142.622,-91.370,170.590,37.320,157.030
C08507=1045.117,142.871,-91.391,170.593,37.322,157.030
C08508=1045.122,143.119,-91.412,170.595,37.323,157.031
C08509=1045.129,143.368,-91.434,170.596,37.325,157.031
C08510=1045.135,143.618,-91.456,170.598,37.326,157.031
C08511=1045.141,143.867,-91.477,170.601,37.327,157.032
C08512=1045.147,144.116,-91.499,170.603,37.329,157.032
C08513=1045.153,144.365,-91.520,170.605,37.330,157.032
C08514=1045.159,144.614,-91.542,170.607,37.332,157.033
C08515=1045.165,144.863,-91.564,170.609,37.333,157.033
C08516=1045.171,145.112,-91.585,170.612,37.335,157.033
C08517=1045.178,145.361,-91.608,170.613,37.337,157.033
C08518=1045.183,145.609,-91.629,170.615,37.338,157.034
C08519=1045.189,145.858,-91.650,170.617,37.340,157.034
C08520=1045.196,146.108,-91.672,170.620,37.341,157.034
C08521=1045.202,146.357,-91.694,170.622,37.343,157.035
C08522=1045.208,146.606,-91.715,170.624,37.344,157.035
C08523=1045.214,146.855,-91.738,170.626,37.345,157.035
C08524=1045.220,147.104,-91.759,170.628,37.347,157.036
C08525=1045.226,147.352,-91.781,170.631,37.348,157.036
C08526=1045.232,147.602,-91.802,170.633,37.350,157.036
C08527=1045.238,147.851,-91.824,170.634,37.351,157.036
C08528=1045.245,148.099,-91.846,170.636,37.353,157.037
C08529=1045.251,148.349,-91.868,170.639,37.354,157.037
C08530=1045.257,148.598,-91.890,170.641,37.356,157.038
C08531=1045.263,148.846,-91.911,170.643,37.357,157.038
C08532=1045.268,149.095,-91.934,170.645,37.359,157.038
C08533=1045.275,149.344,-91.955,170.647,37.360,157.038
C08534=1045.281,149.594,-91.977,170.650,37.362,157.039
C08535=1045.287,149.842,-91.999,170.652,37.363,157.039
C08536=1045.293,150.091,-92.021,170.654,37.365,157.039
C08537=1045.300,150.341,-92.043,170.656,37.367,157.040
C08538=1045.305,150.590,-92.066,170.658,37.368,157.040
C08539=1045.311,150.838,-92.087,170.660,37.370,157.040
C08540=1045.317,151.087,-92.108,170.662,37.371,157.041
C08541=1045.324,151.336,-92.131,170.664,37.373,157.041
C08542=1045.329,151.585,-92.153,170.667,37.374,157.041
C08543=1045.335,151.834,-92.175,170.669,37.376,157.042
C08544=1045.342,152.083,-92.197,170.671,37.377,157.042
C08545=1045.348,152.332,-92.219,170.673,37.379,157.042
C08546=1045.354,152.581,-92.241,170.675,37.380,157.043
C08547=1045.360,152.830,-92.263,170.678,37.382,157.043
C08548=1045.366,153.079,-92.286,170.680,37.383,157.043
C08549=1045.372,153.328,-92.307,170.682,37.385,157.044
C08550=1045.378,153.576,-92.329,170.684,37.386,157.044
C08551=1045.384,153.826,-92.351,170.687,37.388,157.044
C08552=1045.390,154.074,-92.374,170.688,37.390,157.045
C08553=1045.396,154.323,-92.395,170.690,37.391,157.045
C08554=1045.403,154.572,-92.418,170.692,37.393,157.045
C08555=1045.408,154.822,-92.440,170.695,37.394,157.045
C08556=1045.415,155.070,-92.462,170.697,37.396,157.046
C08557=1045.421,155.319,-92.484,170.699,37.397,157.046
C08558=1045.426,155.568,-92.507,170.701,37.398,157.047
C08559=1045.433,155.817,-92.529,170.704,37.400,157.047
C08560=1045.439,156.066,-92.551,170.706,37.401,157.047
C08561=1045.445,156.315,-92.574,170.708,37.403,157.048
C08562=1045.451,156.564,-92.596,170.710,37.405,157.048
C08563=1045.457,156.813,-92.618,170.713,37.406,157.048
C08564=1045.463,157.062,-92.640,170.715,37.408,157.049
C08565=1045.470,157.347,-92.666,170.717,37.410,157.049
C08566=1045.477,157.632,-92.691,170.719,37.412,157.049
C08567=1045.484,157.918,-92.717,170.723,37.414,157.050
C08568=1045.491,158.203,-92.742,170.725,37.415,157.050
C08569=1045.497,158.452,-92.765,170.727,37.416,157.050
C08570=1045.503,158.701,-92.787,170.729,37.418,157.051
C08571=1045.509,158.950,-92.810,170.732,37.420,157.051
C08572=1045.515,159.198,-92.832,170.734,37.421,157.051
C08573=1045.522,159.448,-92.854,170.736,37.423,157.052
C08574=1045.528,159.697,-92.877,170.738,37.424,157.052
C08575=1045.534,159.946,-92.899,170.741,37.426,157.052
C08576=1045.540,160.195,-92.922,170.743,37.428,157.053
C08577=1045.546,160.444,-92.944,170.745,37.429,157.053
C08578=1045.552,160.693,-92.967,170.747,37.431,157.053
C08579=1045.557,160.942,-92.990,170.750,37.433,157.054
C08580=1045.564,161.190,-93.012,170.752,37.434,157.054
C08581=1045.570,161.439,-93.035,170.753,37.436,157.055
C08582=1045.575,161.688,-93.058,170.755,37.438,157.055
C08583=1045.581,161.937,-93.080,170.758,37.439,157.055
C08584=1045.587,162.186,-93.103,170.760,37.441,157.056
C08585=1045.593,162.435,-93.126,170.762,37.443,157.056
C08586=1045.599,162.684,-93.149,170.764,37.445,157.056
C08587=1045.604,162.933,-93.171,170.767,37.447,157.057
C08588=1045.610,163.182,-93.194,170.769,37.448,157.057
C08589=1045.617,163.430,-93.217,170.771,37.450,157.057
C08590=1045.622,163.679,-93.240,170.773,37.451,157.058
C08591=1045.628,163.928,-93.263,170.776,37.453,157.058
C08592=1045.634,164.177,-93.286,170.778,37.455,157.058
C08593=1045.640,164.426,-93.309,170.780,37.457,157.059
C08594=1045.646,164.674,-93.331,170.782,37.458,157.059
C08595=1045.652,164.923,-93.354,170.785,37.460,157.060
C08596=1045.657,165.172,-93.377,170.787,37.462,157.060
C08597=1045.663,165.421,-93.400,170.789,37.463,157.060
C08598=1045.669,165.670,-93.423,170.792,37.465,157.061
C08599=1045.675,165.919,-93.445,170.794,37.467,157.061
C08600=1045.681,166.167,-93.468,170.796,37.468,157.061
C08601=1045.687,166.416,-93.491,170.798,37.470,157.062
C08602=1045.693,166.666,-93.514,170.801,37.472,157.062
C08603=1045.699,166.915,-93.537,170.803,37.473,157.062
C08604=1045.705,167.163,-93.560,170.805,37.475,157.063
C08605=1045.711,167.412,-93.582,170.807,37.477,157.063
C08606=1045.717,167.661,-93.605,170.810,37.478,157.063
C08607=1045.723,167.910,-93.628,170.812,37.480,157.064
C08608=1045.728,168.159,-93.651,170.814,37.482,157.064
C08609=1045.735,168.408,-93.674,170.817,37.484,157.065
C08610=1045.741,168.657,-93.698,170.819,37.485,157.065
C08611=1045.747,168.905,-93.721,170.821,37.487,157.065
C08612=1045.753,169.154,-93.744,170.823,37.488,157.066
C08613=1045.759,169.403,-93.767,170.826,37.490,157.066
C08614=1045.764,169.652,-93.789,170.828,37.492,157.066
C08615=1045.771,169.901,-93.812,170.830,37.494,157.067
C08616=1045.777,170.150,-93.835,170.832,37.496,157.067
C08617=1045.783,170.399,-93.859,170.835,37.497,157.068
C08618=1045.789,170.648,-93.882,170.838,37.499,157.068
C08619=1045.795,170.896,-93.905,170.840,37.500,157.068
C08620=1045.800,171.145,-93.928,170.842,37.502,157.069
C08621=1045.807,171.394,-93.952,170.845,37.504,157.069
C08622=1045.813,171.643,-93.974,170.847,37.506,157.069
C08623=1045.819,171.892,-93.997,170.849,37.508,157.070
C08624=1045.825,172.141,-94.020,170.852,37.509,157.070
C08625=1045.831,172.389,-94.044,170.854,37.511,157.071
C08626=1045.837,172.639,-94.067,170.856,37.512,157.071
C08627=1045.843,172.887,-94.090,170.858,37.514,157.071
C08628=1045.849,173.136,-94.113,170.861,37.516,157.072
C08629=1045.857,173.421,-94.140,170.864,37.518,157.072
C08630=1045.863,173.706,-94.166,170.866,37.520,157.072
C08631=1045.870,173.990,-94.193,170.869,37.522,157.073
C08632=1045.877,174.276,-94.219,170.872,37.524,157.073
C08633=1045.883,174.525,-94.242,170.874,37.525,157.074
C08634=1045.889,174.773,-94.266,170.876,37.527,157.074
C08635=1045.895,175.022,-94.289,170.879,37.529,157.074
C08636=1045.902,175.271,-94.311,170.881,37.531,157.075
C08637=1045.908,175.519,-94.335,170.883,37.533,157.075
C08638=1045.914,175.769,-94.358,170.885,37.534,157.075
C08639=1045.920,176.017,-94.382,170.888,37.536,157.076
C08640=1045.926,176.266,-94.405,170.891,37.537,157.076
C08641=1045.932,176.516,-94.428,170.893,37.539,157.077
C08642=1045.938,176.764,-94.452,170.896,37.541,157.077
C08643=1045.944,177.013,-94.475,170.898,37.543,157.077
C08644=1045.951,177.262,-94.499,170.900,37.545,157.078
C08645=1045.957,177.510,-94.521,170.902,37.546,157.078
C08646=1045.963,177.759,-94.545,170.905,37.548,157.078
C08647=1045.970,178.008,-94.568,170.907,37.549,157.079
C08648=1045.976,178.257,-94.592,170.910,37.551,157.079
C08649=1045.981,178.505,-94.615,170.913,37.553,157.080
C08650=1045.988,178.754,-94.639,170.915,37.555,157.080
C08651=1045.994,179.003,-94.662,170.917,37.556,157.080
C08652=1046.000,179.252,-94.686,170.919,37.558,157.081
C08653=1046.006,179.501,-94.709,170.922,37.560,157.081
C08654=1046.012,179.749,-94.733,170.924,37.562,157.081
C08655=1046.018,179.999,-94.756,170.927,37.564,157.082
C08656=1046.025,180.247,-94.779,170.930,37.565,157.082
C08657=1046.032,180.496,-94.803,170.932,37.566,157.082
C08658=1046.038,180.745,-94.826,170.934,37.568,157.083
C08659=1046.044,180.994,-94.850,170.936,37.570,157.083
C08660=1046.050,181.243,-94.873,170.939,37.572,157.084
C08661=1046.057,181.492,-94.897,170.942,37.574,157.084
C08662=1046.063,181.740,-94.921,170.944,37.575,157.084
C08663=1046.068,181.989,-94.943,170.946,37.577,157.085
C08664=1046.075,182.238,-94.968,170.949,37.579,157.085
C08665=1046.081,182.486,-94.991,170.951,37.581,157.086
C08666=1046.087,182.736,-95.014,170.953,37.583,157.086
C08667=1046.093,182.984,-95.038,170.957,37.584,157.086
C08668=1046.100,183.233,-95.062,170.959,37.586,157.087
C08669=1046.106,183.482,-95.085,170.961,37.587,157.087
C08670=1046.112,183.731,-95.109,170.963,37.589,157.087
C08671=1046.118,183.979,-95.133,170.966,37.591,157.088
C08672=1046.125,184.228,-95.157,170.969,37.593,157.088
C08673=1046.130,184.477,-95.180,170.971,37.595,157.089
C08674=1046.137,184.726,-95.204,170.974,37.597,157.089
C08675=1046.142,184.975,-95.229,170.976,37.599,157.089
C08676=1046.148,185.223,-95.252,170.978,37.601,157.090
C08677=1046.154,185.473,-95.277,170.981,37.603,157.090
C08678=1046.160,185.721,-95.301,170.983,37.604,157.091
C08679=1046.166,185.970,-95.325,170.986,37.606,157.091
C08680=1046.172,186.218,-95.349,170.989,37.609,157.092
C08681=1046.178,186.468,-95.374,170.991,37.610,157.092
C08682=1046.184,186.716,-95.397,170.993,37.612,157.092
C08683=1046.189,186.965,-95.421,170.995,37.614,157.093
C08684=1046.196,187.214,-95.445,170.998,37.616,157.093
C08685=1046.201,187.440,-95.467,171.000,37.618,157.094
C08686=1046.206,187.664,-95.488,171.002,37.619,157.094
C08687=1046.211,187.890,-95.511,171.005,37.621,157.094
C08688=1046.217,188.116,-95.533,171.007,37.623,157.095
C08689=1046.223,188.342,-95.554,171.009,37.625,157.095
C08690=1046.228,188.567,-95.576,171.012,37.626,157.096
C08691=1046.233,188.792,-95.598,171.014,37.628,157.096
C08692=1046.239,189.018,-95.620,171.016,37.630,157.096
C08693=1046.246,189.349,-95.653,171.019,37.632,157.097
C08694=1046.255,189.679,-95.684,171.023,37.635,157.097
C08695=1046.263,190.010,-95.717,171.026,37.638,157.098
C08696=1046.271,190.342,-95.749,171.030,37.641,157.099
C08697=1046.277,190.590,-95.773,171.032,37.642,157.099
C08698=1046.283,190.839,-95.798,171.034,37.644,157.099
C08699=1046.289,191.087,-95.822,171.038,37.646,157.100
C08700=1046.295,191.337,-95.846,171.040,37.648,157.100
C08701=1046.301,191.585,-95.870,171.042,37.650,157.101
C08702=1046.307,191.834,-95.895,171.045,37.652,157.101
C08703=1046.313,192.083,-95.919,171.048,37.654,157.102
C08704=1046.319,192.331,-95.944,171.050,37.656,157.102
C08705=1046.325,192.580,-95.968,171.053,37.658,157.102
C08706=1046.331,192.829,-95.992,171.055,37.660,157.103
C08707=1046.337,193.078,-96.016,171.058,37.662,157.103
C08708=1046.343,193.326,-96.040,171.061,37.664,157.104
C08709=1046.349,193.575,-96.065,171.063,37.666,157.104
C08710=1046.356,193.824,-96.089,171.065,37.668,157.105
C08711=1046.361,194.073,-96.114,171.069,37.670,157.105
C08712=1046.368,194.322,-96.138,171.071,37.671,157.105
C08713=1046.374,194.570,-96.163,171.073,37.674,157.106
C08714=1046.380,194.818,-96.187,171.076,37.676,157.106
C08715=1046.386,195.068,-96.211,171.079,37.677,157.107
C08716=1046.392,195.316,-96.237,171.081,37.680,157.107
C08717=1046.398,195.565,-96.260,171.084,37.682,157.108
C08718=1046.404,195.814,-96.285,171.086,37.683,157.108
C08719=1046.411,196.062,-96.310,171.089,37.686,157.109
C08720=1046.416,196.311,-96.334,171.092,37.687,157.109
C08721=1046.423,196.560,-96.358,171.094,37.689,157.109
C08722=1046.429,196.809,-96.383,171.097,37.692,157.110
C08723=1046.435,197.057,-96.407,171.100,37.693,157.110
C08724=1046.441,197.306,-96.432,171.102,37.695,157.111
C08725=1046.447,197.555,-96.457,171.105,37.697,157.111
C08726=1046.454,197.804,-96.481,171.108,37.699,157.111
C08727=1046.459,198.052,-96.506,171.110,37.702,157.112
C08728=1046.466,198.301,-96.530,171.112,37.703,157.112
C08729=1046.472,198.549,-96.555,171.116,37.705,157.113
C08730=1046.478,198.799,-96.580,171.118,37.708,157.113
C08731=1046.485,199.046,-96.604,171.120,37.709,157.114
C08732=1046.490,199.296,-96.629,171.124,37.711,157.114
C08733=1046.497,199.545,-96.653,171.126,37.713,157.115
C08734=1046.503,199.793,-96.678,171.128,37.715,157.115
C08735=1046.510,200.042,-96.703,171.132,37.718,157.116
C08736=1046.516,200.290,-96.727,171.134,37.719,157.116
C08737=1046.522,200.539,-96.753,171.136,37.721,157.116
C08738=1046.528,200.788,-96.777,171.140,37.723,157.117
C08739=1046.535,201.037,-96.802,171.142,37.725,157.117
C08740=1046.540,201.286,-96.827,171.144,37.728,157.118
C08741=1046.547,201.533,-96.851,171.148,37.729,157.118
C08742=1046.553,201.783,-96.876,171.150,37.732,157.119
C08743=1046.559,202.031,-96.901,171.152,37.733,157.119
C08744=1046.565,202.280,-96.926,171.156,37.736,157.120
C08745=1046.571,202.529,-96.951,171.158,37.738,157.120
C08746=1046.577,202.777,-96.976,171.161,37.740,157.120
C08747=1046.583,203.026,-97.001,171.164,37.742,157.121
C08748=1046.589,203.275,-97.027,171.166,37.744,157.121
C08749=1046.595,203.524,-97.051,171.169,37.746,157.122
C08750=1046.601,203.773,-97.077,171.172,37.749,157.122
C08751=1046.607,204.021,-97.102,171.174,37.751,157.123
C08752=1046.614,204.269,-97.126,171.177,37.753,157.123
C08753=1046.620,204.518,-97.151,171.180,37.755,157.124
C08754=1046.626,204.767,-97.176,171.182,37.757,157.124
C08755=1046.632,205.016,-97.202,171.186,37.759,157.125
C08756=1046.638,205.264,-97.227,171.188,37.761,157.125
C08757=1046.664,206.316,-97.333,171.438,37.861,157.149
C08758=1046.671,206.588,-97.362,171.440,37.864,157.150
C08759=1046.678,206.858,-97.390,171.443,37.867,157.151
C08760=1046.685,207.130,-97.418,171.444,37.871,157.151
C08761=1046.692,207.401,-97.448,171.447,37.874,157.152
C08762=1046.699,207.650,-97.473,171.448,37.877,157.153
C08763=1046.706,207.898,-97.500,171.451,37.880,157.153
C08764=1046.711,208.147,-97.526,171.453,37.883,157.154
C08765=1046.718,208.395,-97.553,171.455,37.886,157.155
C08766=1046.725,208.643,-97.579,171.457,37.888,157.155
C08767=1046.731,208.892,-97.606,171.459,37.891,157.156
C08768=1046.738,209.140,-97.632,171.461,37.894,157.157
C08769=1046.745,209.389,-97.658,171.463,37.897,157.157
C08770=1046.751,209.637,-97.684,171.465,37.900,157.158
C08771=1046.758,209.886,-97.711,171.467,37.903,157.159
C08772=1046.764,210.134,-97.737,171.469,37.906,157.159
C08773=1046.770,210.384,-97.764,171.472,37.909,157.160
C08774=1046.777,210.632,-97.790,171.473,37.912,157.160
C08775=1046.784,210.881,-97.816,171.476,37.915,157.161
C08776=1046.790,211.129,-97.843,171.477,37.917,157.162
C08777=1046.797,211.378,-97.869,171.480,37.920,157.162
C08778=1046.803,211.626,-97.896,171.482,37.923,157.163
C08779=1046.810,211.875,-97.922,171.484,37.926,157.164
C08780=1046.817,212.123,-97.949,171.486,37.929,157.164
C08781=1046.823,212.372,-97.976,171.488,37.932,157.165
C08782=1046.829,212.620,-98.003,171.491,37.935,157.166
C08783=1046.836,212.869,-98.029,171.492,37.938,157.166
C08784=1046.842,213.117,-98.056,171.495,37.941,157.167
C08785=1046.849,213.366,-98.082,171.497,37.944,157.168
C08786=1046.855,213.614,-98.109,171.499,37.947,157.168
C08787=1046.862,213.863,-98.135,171.501,37.949,157.169
C08788=1046.867,214.111,-98.162,171.503,37.952,157.169
C08789=1046.875,214.359,-98.189,171.505,37.955,157.170
C08790=1046.881,214.608,-98.216,171.508,37.958,157.171
C08791=1046.887,214.857,-98.243,171.509,37.961,157.171
C08792=1046.894,215.105,-98.269,171.512,37.964,157.172
C08793=1046.900,215.354,-98.296,171.514,37.967,157.173
C08794=1046.907,215.601,-98.322,171.516,37.970,157.173
C08795=1046.913,215.850,-98.349,171.518,37.973,157.174
C08796=1046.920,216.099,-98.376,171.520,37.975,157.174
C08797=1046.926,216.348,-98.403,171.522,37.978,157.175
C08798=1046.932,216.597,-98.430,171.525,37.981,157.176
C08799=1046.939,216.844,-98.456,171.526,37.984,157.176
C08800=1046.946,217.093,-98.483,171.529,37.987,157.177
C08801=1046.953,217.342,-98.510,171.531,37.990,157.178
C08802=1046.959,217.590,-98.537,171.533,37.993,157.178
C08803=1046.965,217.839,-98.564,171.535,37.995,157.179
C08804=1046.972,218.087,-98.590,171.538,37.998,157.180
C08805=1046.978,218.336,-98.617,171.539,38.001,157.180
C08806=1046.985,218.584,-98.644,171.542,38.004,157.181
C08807=1046.991,218.832,-98.671,171.544,38.007,157.181
C08808=1046.998,219.081,-98.697,171.546,38.010,157.182
C08809=1047.005,219.329,-98.725,171.548,38.012,157.183
C08810=1047.011,219.578,-98.752,171.551,38.015,157.183
C08811=1047.018,219.826,-98.779,171.552,38.018,157.184
C08812=1047.025,220.075,-98.806,171.555,38.021,157.185
C08813=1047.031,220.323,-98.832,171.557,38.024,157.185
C08814=1047.039,220.600,-98.862,171.560,38.027,157.186
C08815=1047.045,220.877,-98.894,171.563,38.031,157.187
C08816=1047.052,221.153,-98.923,171.564,38.034,157.187
C08817=1047.060,221.430,-98.954,171.567,38.037,157.188
C08818=1047.065,221.679,-98.980,171.569,38.040,157.189
C08819=1047.073,221.927,-99.008,171.572,38.043,157.189
C08820=1047.079,222.176,-99.035,171.573,38.046,157.190
C08821=1047.085,222.424,-99.062,171.576,38.048,157.191
C08822=1047.092,222.673,-99.089,171.578,38.051,157.191
C08823=1047.098,222.921,-99.117,171.581,38.054,157.192
C08824=1047.104,223.169,-99.144,171.582,38.057,157.193
C08825=1047.111,223.418,-99.171,171.585,38.060,157.193
C08826=1047.118,223.666,-99.198,171.587,38.063,157.194
C08827=1047.124,223.915,-99.225,171.589,38.066,157.194
C08828=1047.131,224.163,-99.253,171.591,38.069,157.195
C08829=1047.137,224.411,-99.280,171.594,38.071,157.196
C08830=1047.144,224.661,-99.307,171.596,38.074,157.196
C08831=1047.150,224.908,-99.335,171.598,38.077,157.197
C08832=1047.156,225.157,-99.362,171.600,38.080,157.198
C08833=1047.163,225.406,-99.389,171.603,38.083,157.198
C08834=1047.170,225.653,-99.416,171.605,38.086,157.199
C08835=1047.176,225.902,-99.443,171.607,38.089,157.200
C08836=1047.183,226.151,-99.471,171.610,38.092,157.200
C08837=1047.189,226.399,-99.499,171.612,38.094,157.201
C08838=1047.196,226.648,-99.526,171.615,38.097,157.201
C08839=1047.202,226.896,-99.553,171.616,38.100,157.202
C08840=1047.209,227.144,-99.581,171.619,38.103,157.203
C08841=1047.215,227.393,-99.608,171.621,38.106,157.203
C08842=1047.222,227.642,-99.635,171.624,38.109,157.204
C08843=1047.228,227.889,-99.662,171.626,38.111,157.205
C08844=1047.235,228.138,-99.690,171.628,38.114,157.205
C08845=1047.242,228.386,-99.718,171.630,38.117,157.206
C08846=1047.249,228.635,-99.745,171.633,38.120,157.207
C08847=1047.255,228.884,-99.772,171.635,38.123,157.207
C08848=1047.262,229.132,-99.800,171.637,38.125,157.208
C08849=1047.268,229.380,-99.828,171.639,38.128,157.208
C08850=1047.274,229.628,-99.855,171.642,38.131,157.209
C08851=1047.281,229.877,-99.883,171.644,38.134,157.210
C08852=1047.287,230.125,-99.911,171.647,38.137,157.210
C08853=1047.294,230.374,-99.939,171.648,38.140,157.211
C08854=1047.299,230.622,-99.966,171.651,38.143,157.212
C08855=1047.306,230.871,-99.993,171.653,38.145,157.212
C08856=1047.313,231.119,-100.021,171.656,38.148,157.213
C08857=1047.319,231.368,-100.049,171.658,38.151,157.214
C08858=1047.326,231.616,-100.077,171.660,38.154,157.214
C08859=1047.333,231.865,-100.104,171.663,38.157,157.215
C08860=1047.338,232.113,-100.132,171.665,38.160,157.216
C08861=1047.345,232.361,-100.160,171.668,38.163,157.216
C08862=1047.352,232.609,-100.188,171.670,38.165,157.217
C08863=1047.358,232.858,-100.216,171.673,38.168,157.217
C08864=1047.365,233.106,-100.243,171.674,38.171,157.218
C08865=1047.371,233.355,-100.272,171.677,38.174,157.219
C08866=1047.377,233.603,-100.299,171.679,38.177,157.219
C08867=1047.384,233.851,-100.327,171.682,38.180,157.220
C08868=1047.391,234.099,-100.355,171.684,38.183,157.221
C08869=1047.397,234.348,-100.383,171.687,38.185,157.221
C08870=1047.402,234.559,-100.407,171.688,38.188,157.222
C08871=1047.408,234.769,-100.431,171.691,38.190,157.223
C08872=1047.413,234.980,-100.454,171.692,38.193,157.223
C08873=1047.419,235.191,-100.478,171.695,38.195,157.224
C08874=1047.424,235.402,-100.502,171.696,38.197,157.224
C08875=1047.429,235.611,-100.525,171.699,38.200,157.225
C08876=1047.435,235.822,-100.549,171.701,38.202,157.225
C08877=1047.441,236.033,-100.573,171.702,38.204,157.226
C08878=1047.447,236.281,-100.601,171.705,38.207,157.226
C08879=1047.453,236.530,-100.629,171.708,38.210,157.227
C08880=1047.460,236.778,-100.657,171.710,38.213,157.228
C08881=1047.467,237.027,-100.684,171.713,38.216,157.228
C08882=1047.473,237.275,-100.713,171.714,38.219,157.229
C08883=1047.480,237.523,-100.741,171.717,38.222,157.230
C08884=1047.486,237.772,-100.769,171.719,38.224,157.230
C08885=1047.493,238.020,-100.797,171.722,38.227,157.231
C08886=1047.502,238.365,-100.836,171.726,38.231,157.232
C08887=1047.511,238.709,-100.875,171.728,38.235,157.233
C08888=1047.520,239.054,-100.915,171.732,38.239,157.234
C08889=1047.529,239.399,-100.953,171.736,38.243,157.235
C08890=1047.535,239.647,-100.981,171.738,38.246,157.235
C08891=1047.542,239.895,-101.010,171.741,38.249,157.236
C08892=1047.548,240.144,-101.038,171.742,38.251,157.236
C08893=1047.555,240.392,-101.067,171.745,38.254,157.237
C08894=1047.561,240.640,-101.095,171.747,38.257,157.238
C08895=1047.568,240.889,-101.122,171.750,38.260,157.238
C08896=1047.574,241.137,-101.151,171.753,38.263,157.239
C08897=1047.581,241.385,-101.179,171.755,38.266,157.240
C08898=1047.587,241.633,-101.208,171.758,38.268,157.240
C08899=1047.594,241.882,-101.236,171.760,38.271,157.241
C08900=1047.600,242.130,-101.265,171.763,38.274,157.242
C08901=1047.607,242.378,-101.293,171.765,38.277,157.242
C08902=1047.613,242.626,-101.322,171.768,38.279,157.243
C08903=1047.619,242.875,-101.350,171.770,38.282,157.244
C08904=1047.626,243.123,-101.378,171.773,38.285,157.244
C08905=1047.632,243.372,-101.407,171.776,38.288,157.245
C08906=1047.639,243.620,-101.435,171.778,38.291,157.246
C08907=1047.645,243.869,-101.464,171.781,38.294,157.246
C08908=1047.652,244.117,-101.493,171.782,38.296,157.247
C08909=1047.659,244.365,-101.521,171.785,38.299,157.247
C08910=1047.665,244.614,-101.550,171.787,38.302,157.248
C08911=1047.671,244.862,-101.578,171.790,38.305,157.249
C08912=1047.678,245.110,-101.607,171.792,38.308,157.249
C08913=1047.684,245.358,-101.635,171.795,38.311,157.250
C08914=1047.691,245.606,-101.664,171.797,38.314,157.251
C08915=1047.697,245.854,-101.693,171.800,38.317,157.252
C08916=1047.703,246.103,-101.721,171.803,38.320,157.252
C08917=1047.709,246.351,-101.750,171.805,38.323,157.253
C08918=1047.715,246.599,-101.779,171.808,38.325,157.254
C08919=1047.722,246.847,-101.808,171.810,38.328,157.254
C08920=1047.728,247.096,-101.836,171.813,38.331,157.255
C08921=1047.735,247.344,-101.865,171.815,38.334,157.256
C08922=1047.741,247.593,-101.895,171.818,38.337,157.256
C08923=1047.748,247.841,-101.924,171.821,38.340,157.257
C08924=1047.754,248.089,-101.953,171.823,38.343,157.258
C08925=1047.760,248.338,-101.981,171.826,38.345,157.258
C08926=1047.767,248.601,-102.012,171.828,38.349,157.259
C08927=1047.774,248.864,-102.042,171.831,38.352,157.260
C08928=1047.780,249.127,-102.073,171.833,38.355,157.260
C08929=1047.787,249.391,-102.103,171.837,38.358,157.261
C08930=1047.794,249.639,-102.132,171.840,38.361,157.262
C08931=1047.800,249.888,-102.161,171.842,38.363,157.262
C08932=1047.806,250.136,-102.190,171.845,38.366,157.263
C08933=1047.813,250.385,-102.220,171.847,38.369,157.264
C08934=1047.819,250.633,-102.249,171.850,38.372,157.264
C08935=1047.825,250.881,-102.278,171.852,38.375,157.265
C08936=1047.832,251.129,-102.306,171.855,38.378,157.266
C08937=1047.839,251.377,-102.335,171.858,38.381,157.266
C08938=1047.845,251.626,-102.365,171.860,38.384,157.267
C08939=1047.852,251.874,-102.394,171.863,38.386,157.268
C08940=1047.858,252.122,-102.423,171.865,38.389,157.268
C08941=1047.864,252.370,-102.452,171.868,38.392,157.269
C08942=1047.870,252.618,-102.481,171.870,38.395,157.270
C08943=1047.877,252.867,-102.510,171.873,38.398,157.270
C08944=1047.884,253.115,-102.539,171.876,38.401,157.271
C08945=1047.890,253.363,-102.568,171.878,38.404,157.272
C08946=1047.897,253.611,-102.597,171.881,38.407,157.272
C08947=1047.904,253.860,-102.626,171.883,38.409,157.273
C08948=1047.910,254.108,-102.655,171.887,38.412,157.274
C08949=1047.916,254.356,-102.685,171.889,38.415,157.274
C08950=1047.923,254.604,-102.714,171.892,38.418,157.275
C08951=1047.930,254.852,-102.743,171.895,38.421,157.276
C08952=1047.936,255.101,-102.773,171.897,38.423,157.276
C08953=1047.942,255.349,-102.802,171.900,38.426,157.277
C08954=1047.948,255.597,-102.831,171.902,38.429,157.278
C08955=1047.955,255.845,-102.861,171.905,38.432,157.278
C08956=1047.962,256.093,-102.890,171.907,38.435,157.279
C08957=1047.968,256.341,-102.919,171.910,38.438,157.280
C08958=1047.975,256.590,-102.948,171.914,38.441,157.280
C08959=1047.981,256.838,-102.977,171.916,38.443,157.281
C08960=1047.988,257.086,-103.006,171.919,38.446,157.282
C08961=1047.995,257.334,-103.036,171.921,38.449,157.282
C08962=1048.001,257.582,-103.065,171.924,38.452,157.283
C08963=1048.008,257.830,-103.095,171.926,38.455,157.284
C08964=1048.015,258.079,-103.124,171.929,38.457,157.284
C08965=1048.021,258.327,-103.153,171.933,38.460,157.285
C08966=1048.028,258.576,-103.182,171.935,38.463,157.286
C08967=1048.035,258.823,-103.212,171.938,38.466,157.286
C08968=1048.041,259.071,-103.241,171.940,38.469,157.287
C08969=1048.048,259.320,-103.271,171.943,38.471,157.288
C08970=1048.054,259.568,-103.300,171.945,38.474,157.288
C08971=1048.061,259.817,-103.330,171.949,38.477,157.289
C08972=1048.068,260.064,-103.360,171.952,38.480,157.290
C08973=1048.074,260.312,-103.389,171.954,38.483,157.290
C08974=1048.081,260.561,-103.418,171.957,38.486,157.291
C08975=1048.087,260.809,-103.448,171.959,38.489,157.292
C08976=1048.094,261.057,-103.477,171.963,38.491,157.292
C08977=1048.101,261.305,-103.507,171.965,38.494,157.293
C08978=1048.108,261.554,-103.536,171.968,38.497,157.294
C08979=1048.114,261.801,-103.566,171.971,38.499,157.294
C08980=1048.121,262.050,-103.596,171.973,38.502,157.295
C08981=1048.127,262.298,-103.625,171.977,38.505,157.296
C08982=1048.134,262.560,-103.656,171.979,38.508,157.296
C08983=1048.141,262.821,-103.687,171.982,38.511,157.297
C08984=1048.148,263.083,-103.718,171.986,38.514,157.298
C08985=1048.155,263.345,-103.751,171.988,38.517,157.298
C08986=1048.162,263.594,-103.780,171.991,38.520,157.299
C08987=1048.168,263.842,-103.811,171.993,38.523,157.300
C08988=1048.175,264.090,-103.841,171.996,38.526,157.300
C08989=1048.181,264.338,-103.870,172.000,38.529,157.301
C08990=1048.188,264.587,-103.900,172.002,38.532,157.302
C08991=1048.194,264.834,-103.930,172.005,38.534,157.303
C08992=1048.201,265.082,-103.960,172.007,38.537,157.303
C08993=1048.207,265.331,-103.990,172.011,38.541,157.304
C08994=1048.213,265.578,-104.020,172.014,38.544,157.305
C08995=1048.220,265.826,-104.050,172.016,38.546,157.305
C08996=1048.226,266.074,-104.080,172.019,38.549,157.306
C08997=1048.233,266.323,-104.110,172.021,38.552,157.307
C08998=1048.240,266.571,-104.139,172.025,38.555,157.307
C08999=1048.246,266.819,-104.170,172.028,38.558,157.308
C09000=1048.253,267.067,-104.200,172.030,38.561,157.309
C09001=1048.260,267.315,-104.230,172.033,38.564,157.309
C09002=1048.266,267.564,-104.260,172.036,38.566,157.310
C09003=1048.272,267.812,-104.290,172.039,38.569,157.311
C09004=1048.279,268.060,-104.320,172.042,38.572,157.312
C09005=1048.285,268.308,-104.350,172.045,38.575,157.312
C09006=1048.292,268.556,-104.381,172.048,38.578,157.313
C09007=1048.298,268.804,-104.411,172.050,38.581,157.314
C09008=1048.306,269.052,-104.441,172.053,38.584,157.314
C09009=1048.311,269.300,-104.471,172.057,38.586,157.315
C09010=1048.319,269.548,-104.501,172.059,38.590,157.316
C09011=1048.324,269.796,-104.532,172.062,38.593,157.316
C09012=1048.332,270.044,-104.562,172.064,38.596,157.317
C09013=1048.338,270.292,-104.592,172.068,38.598,157.318
C09014=1048.344,270.540,-104.623,172.071,38.601,157.319
C09015=1048.351,270.788,-104.653,172.073,38.604,157.319
C09016=1048.357,271.036,-104.683,172.077,38.607,157.320
C09017=1048.364,271.284,-104.713,172.079,38.610,157.321
C09018=1048.370,271.533,-104.744,172.082,38.613,157.321
C09019=1048.377,271.781,-104.774,172.086,38.616,157.322
C09020=1048.383,272.029,-104.805,172.088,38.619,157.323
C09021=1048.390,272.277,-104.835,172.091,38.622,157.323
C09022=1048.397,272.524,-104.866,172.094,38.625,157.324
C09023=1048.403,272.773,-104.896,172.097,38.628,157.325
C09024=1048.410,273.020,-104.926,172.100,38.630,157.326
C09025=1048.416,273.269,-104.957,172.102,38.633,157.326
C09026=1048.422,273.518,-104.988,172.106,38.637,157.327
C09027=1048.429,273.764,-105.018,172.109,38.640,157.328
C09028=1048.436,274.013,-105.049,172.111,38.642,157.328
C09029=1048.442,274.261,-105.080,172.115,38.645,157.329
C09030=1048.449,274.509,-105.109,172.118,38.648,157.330
C09031=1048.455,274.757,-105.141,172.120,38.652,157.331
C09032=1048.462,275.005,-105.171,172.124,38.654,157.331
C09033=1048.468,275.253,-105.202,172.126,38.657,157.332
C09034=1048.475,275.501,-105.233,172.129,38.660,157.333
C09035=1048.481,275.749,-105.263,172.133,38.663,157.333
C09036=1048.487,275.997,-105.294,172.135,38.666,157.334
C09037=1048.494,276.245,-105.325,172.139,38.669,157.335
C09038=1048.501,276.512,-105.357,172.142,38.672,157.336
C09039=1048.508,276.778,-105.391,172.145,38.675,157.336
C09040=1048.515,277.043,-105.424,172.148,38.679,157.337
C09041=1048.522,277.310,-105.457,172.152,38.682,157.338
C09042=1048.529,277.558,-105.487,172.154,38.685,157.339
